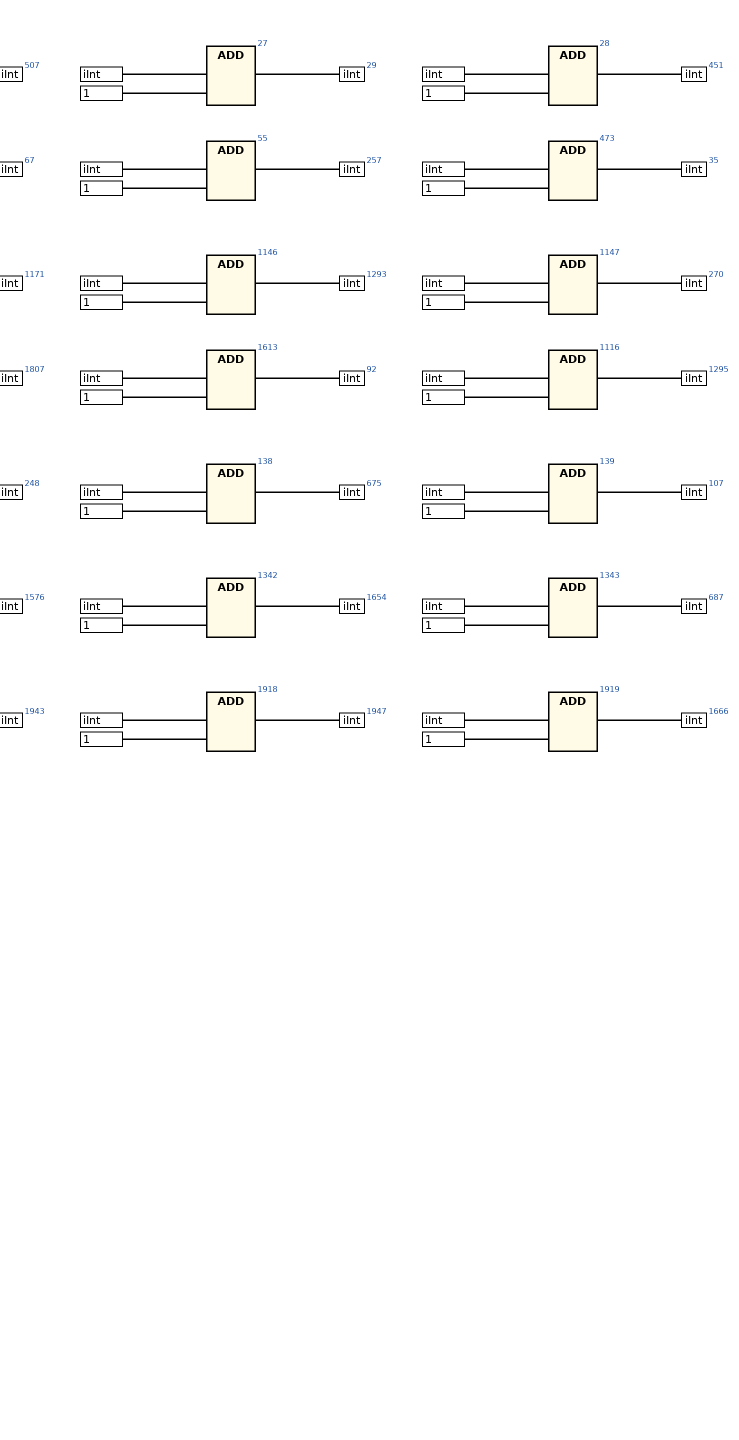
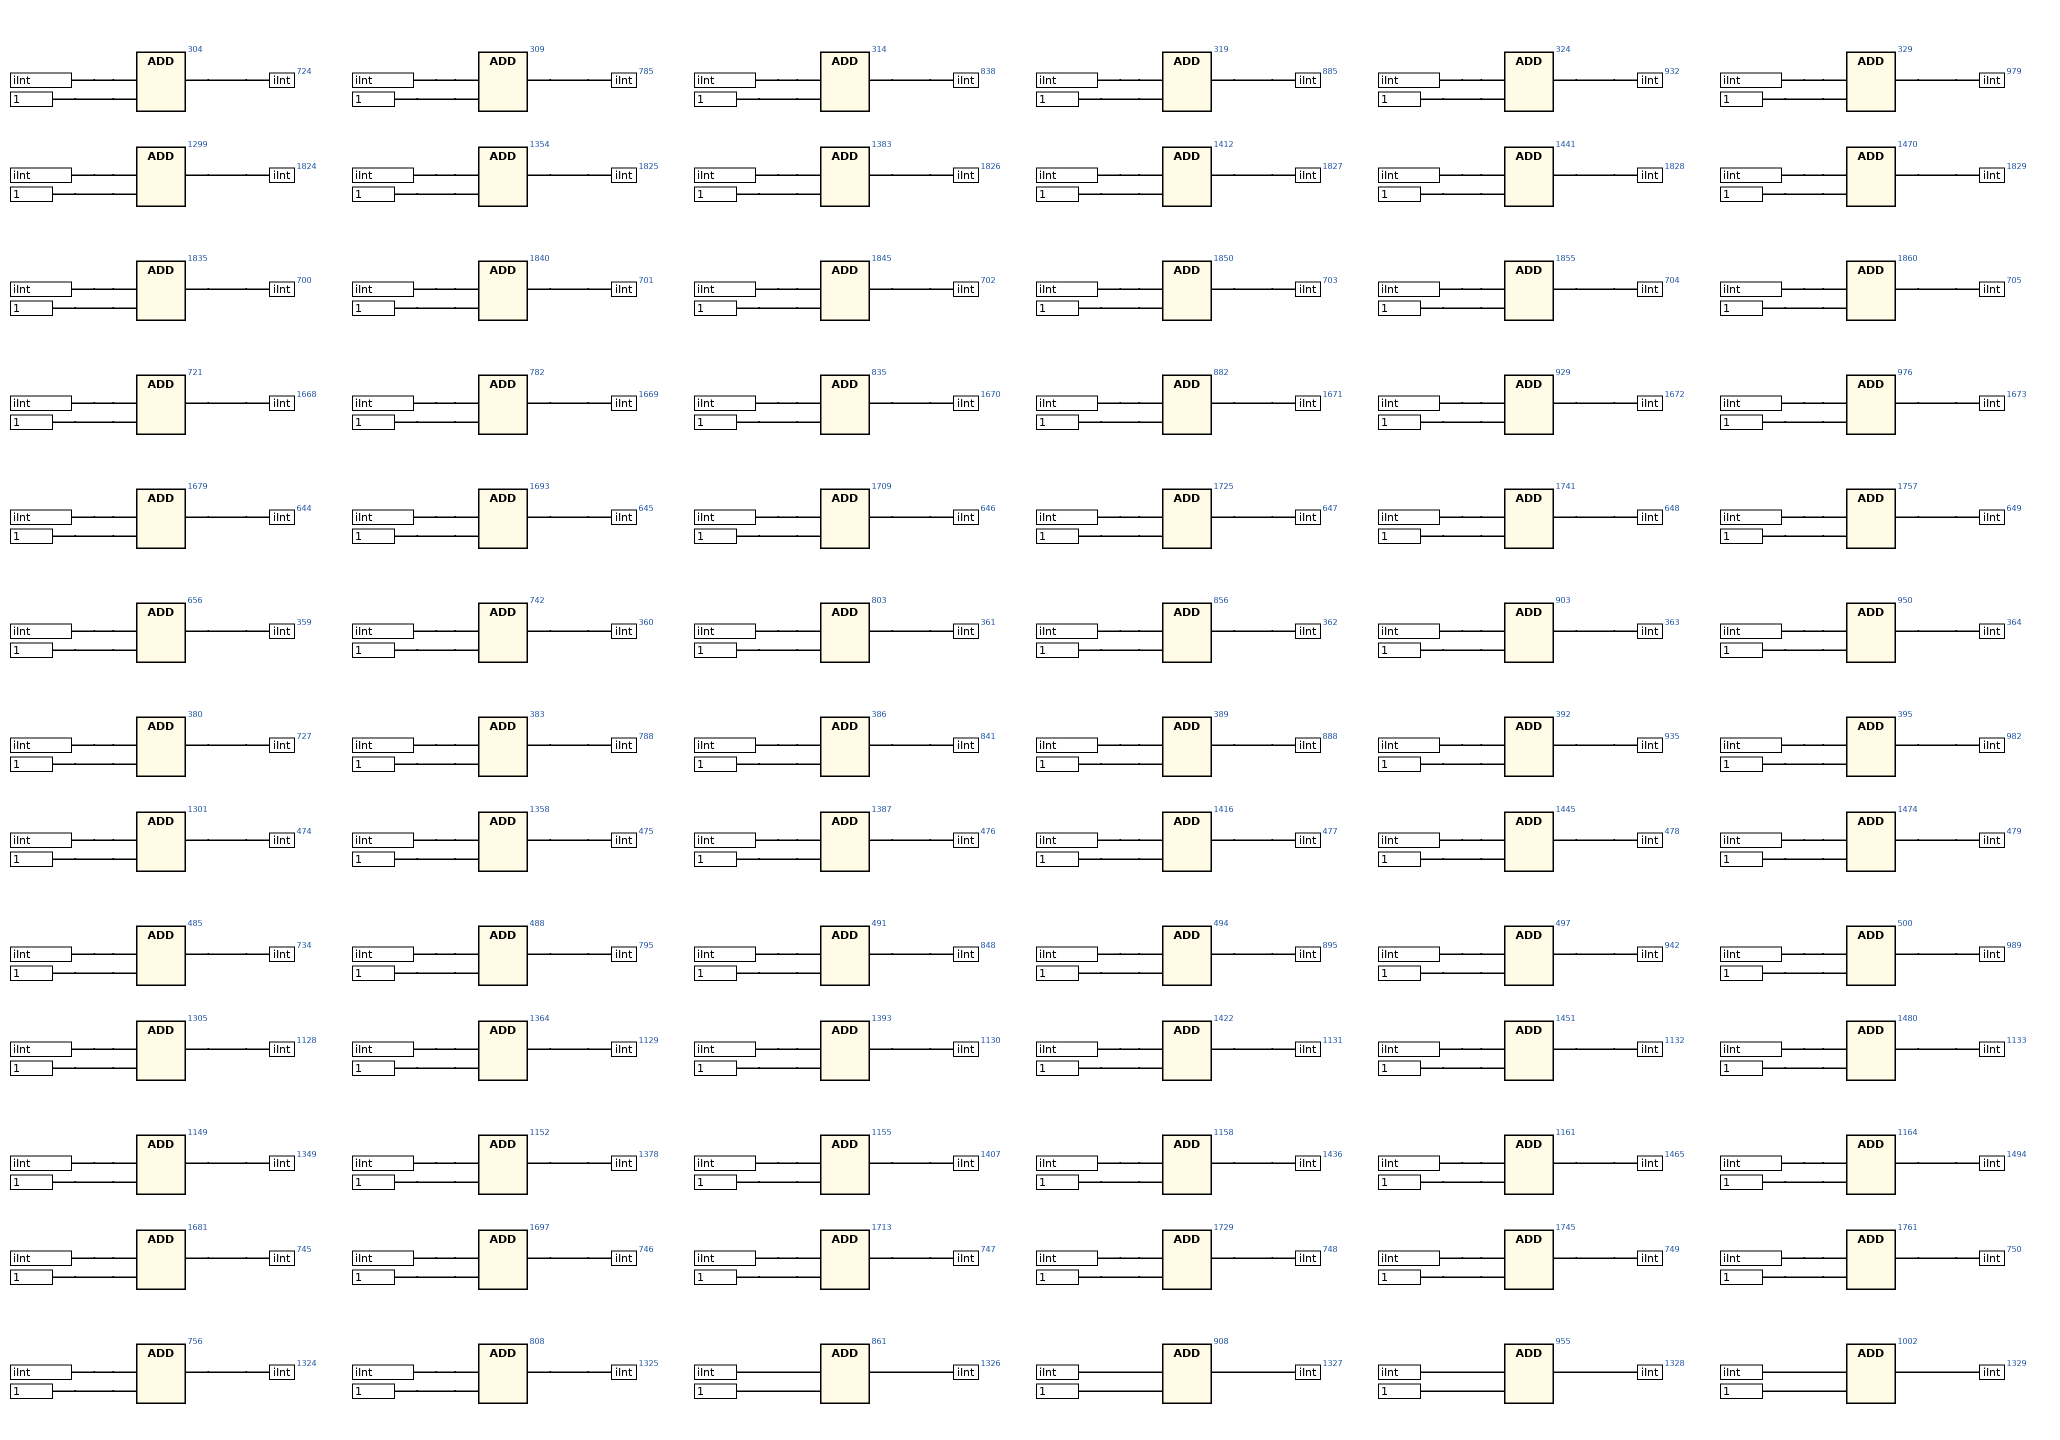
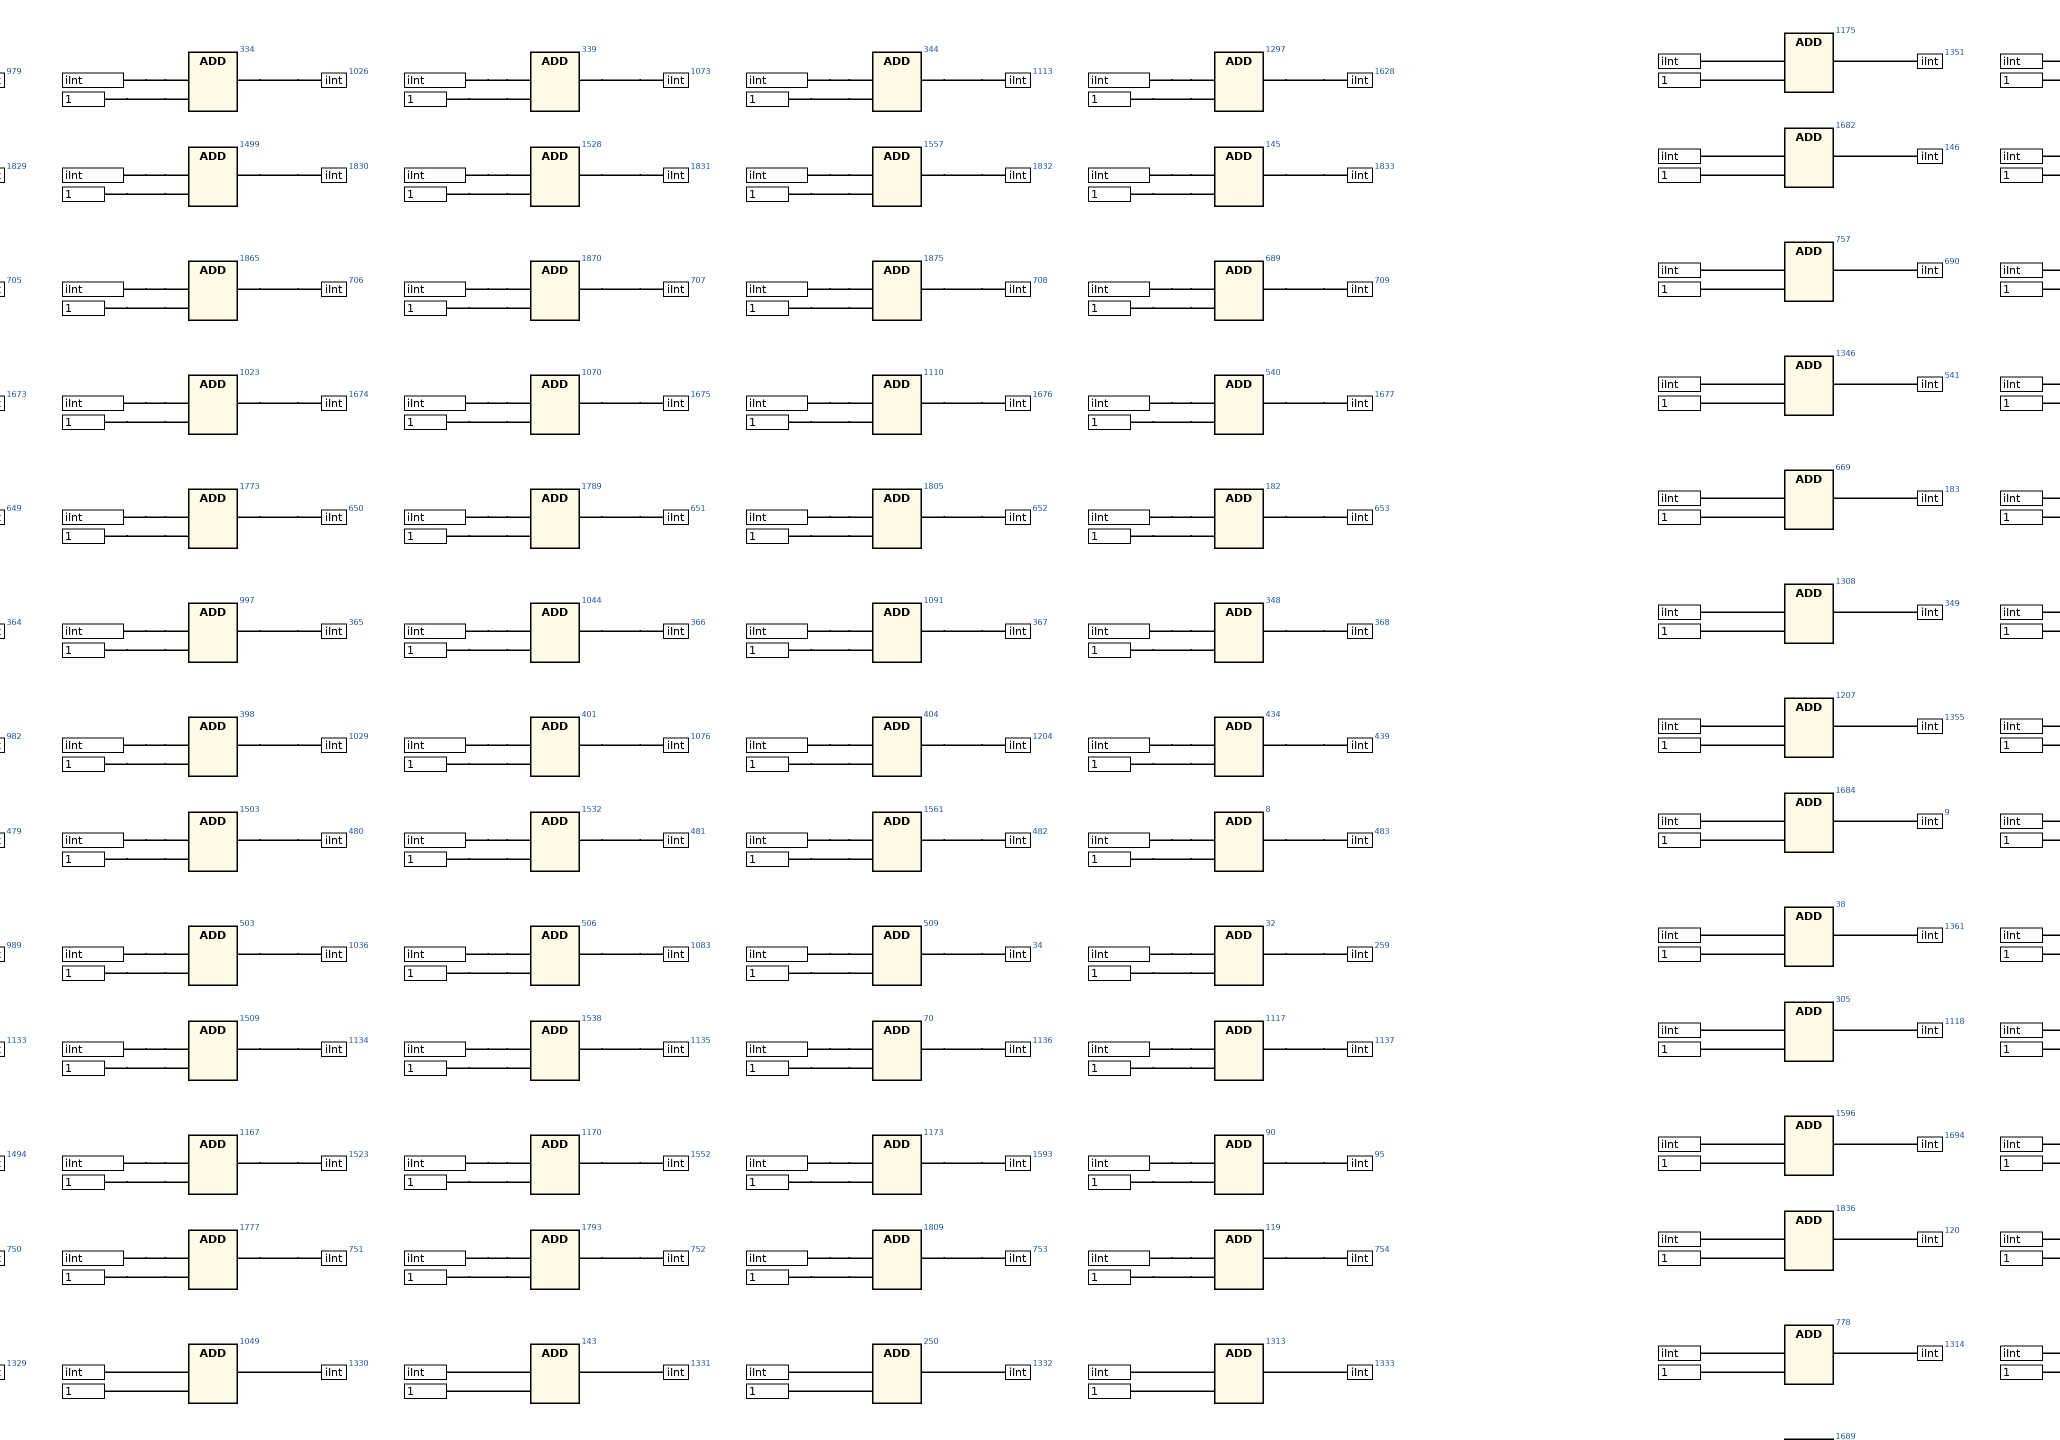
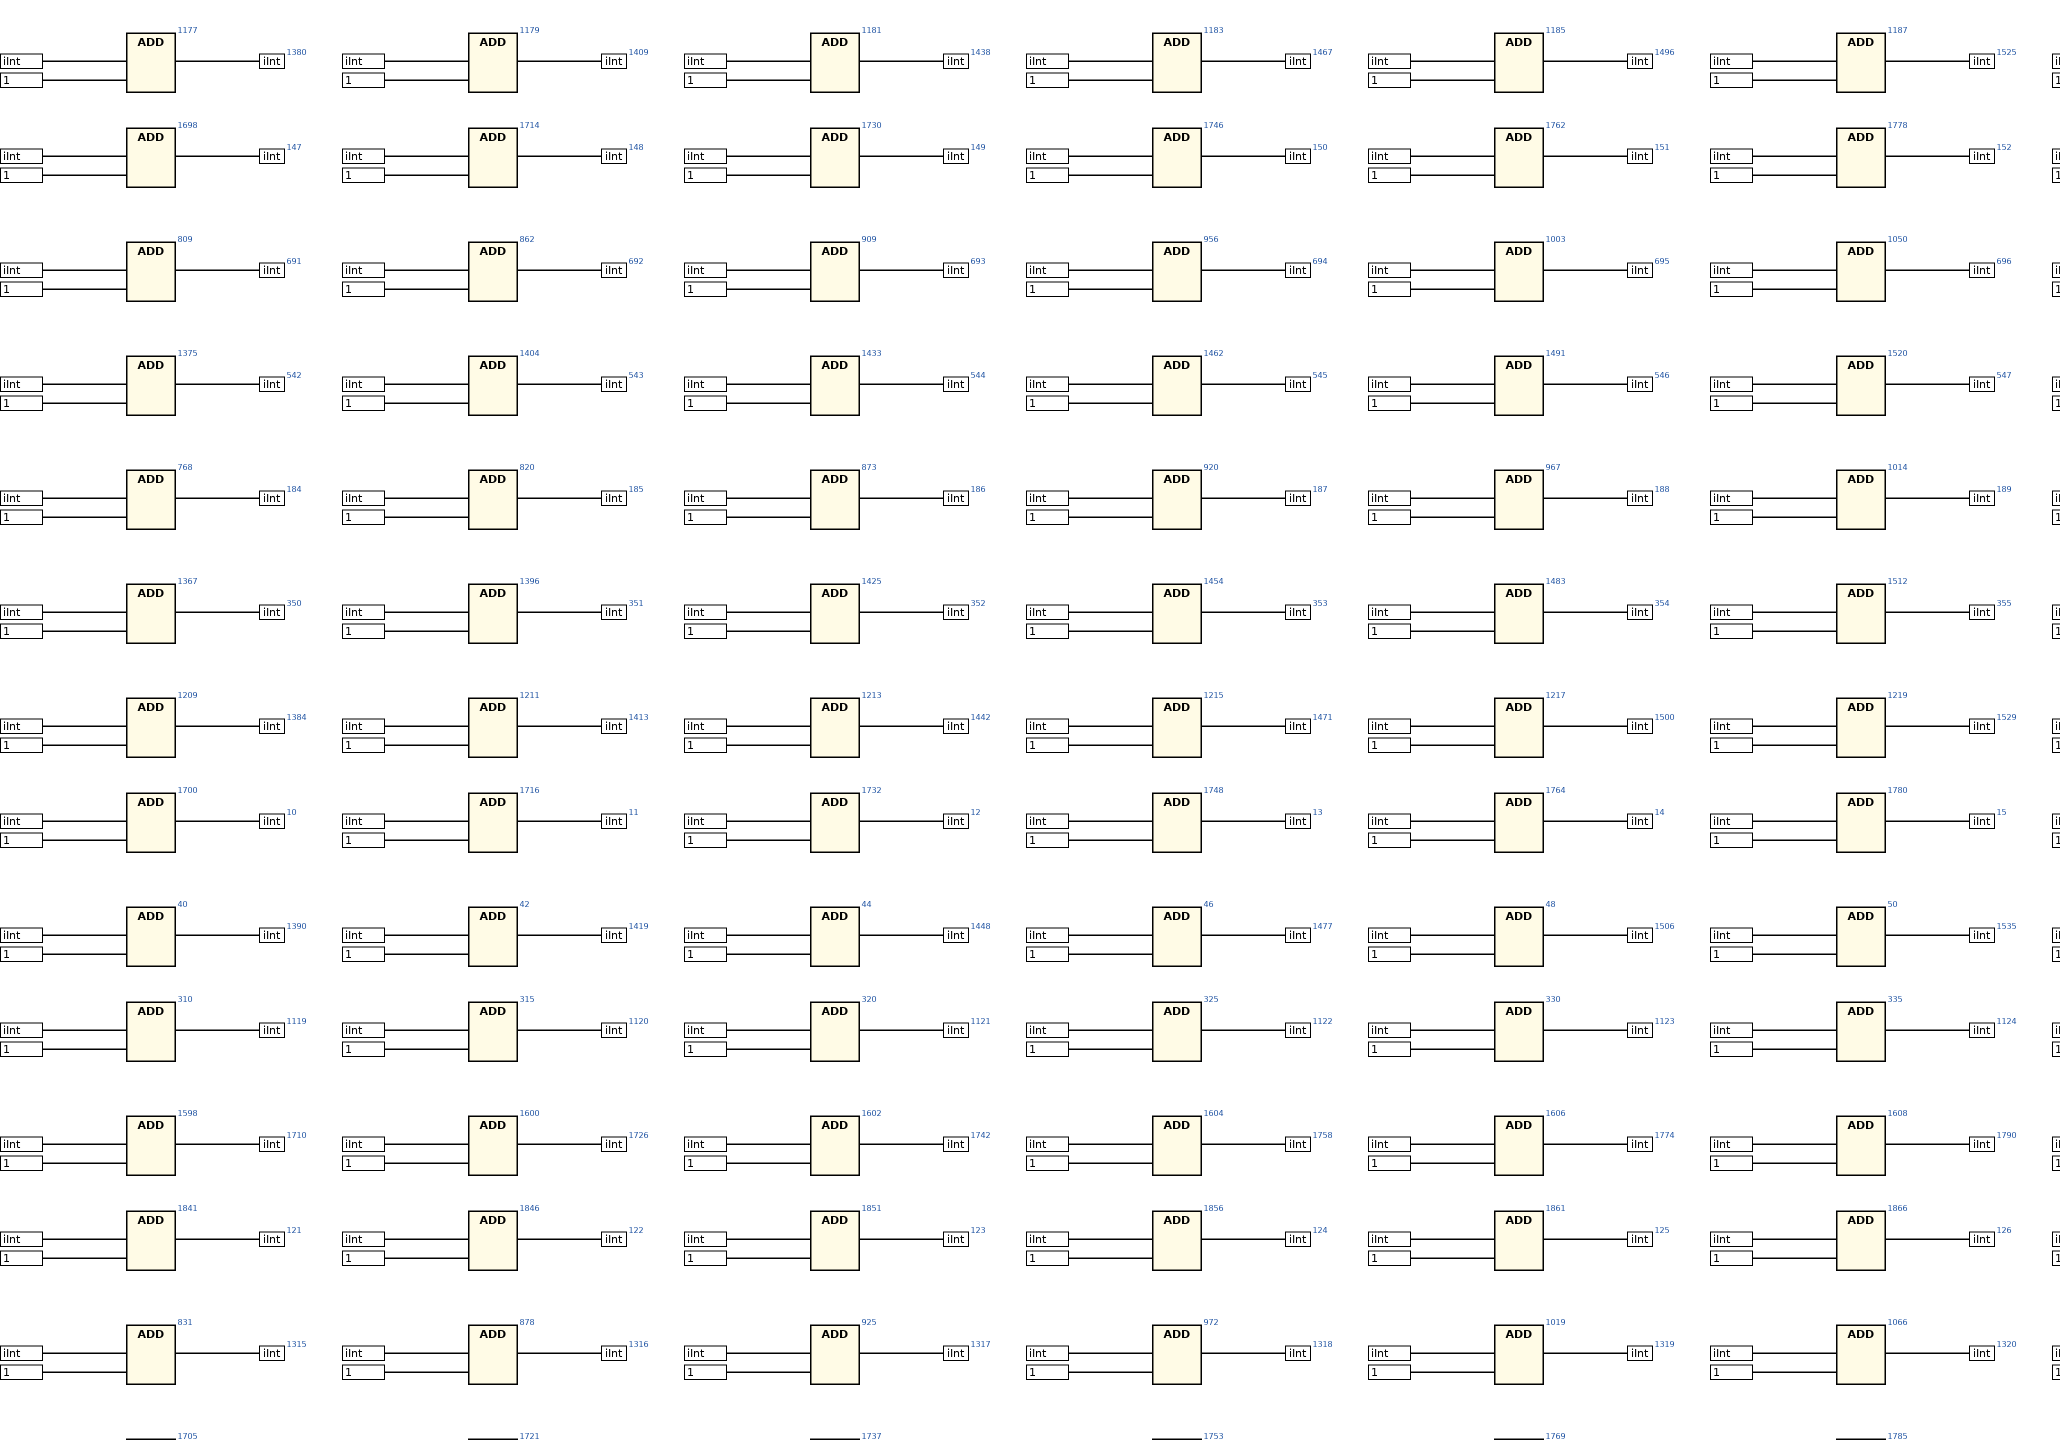
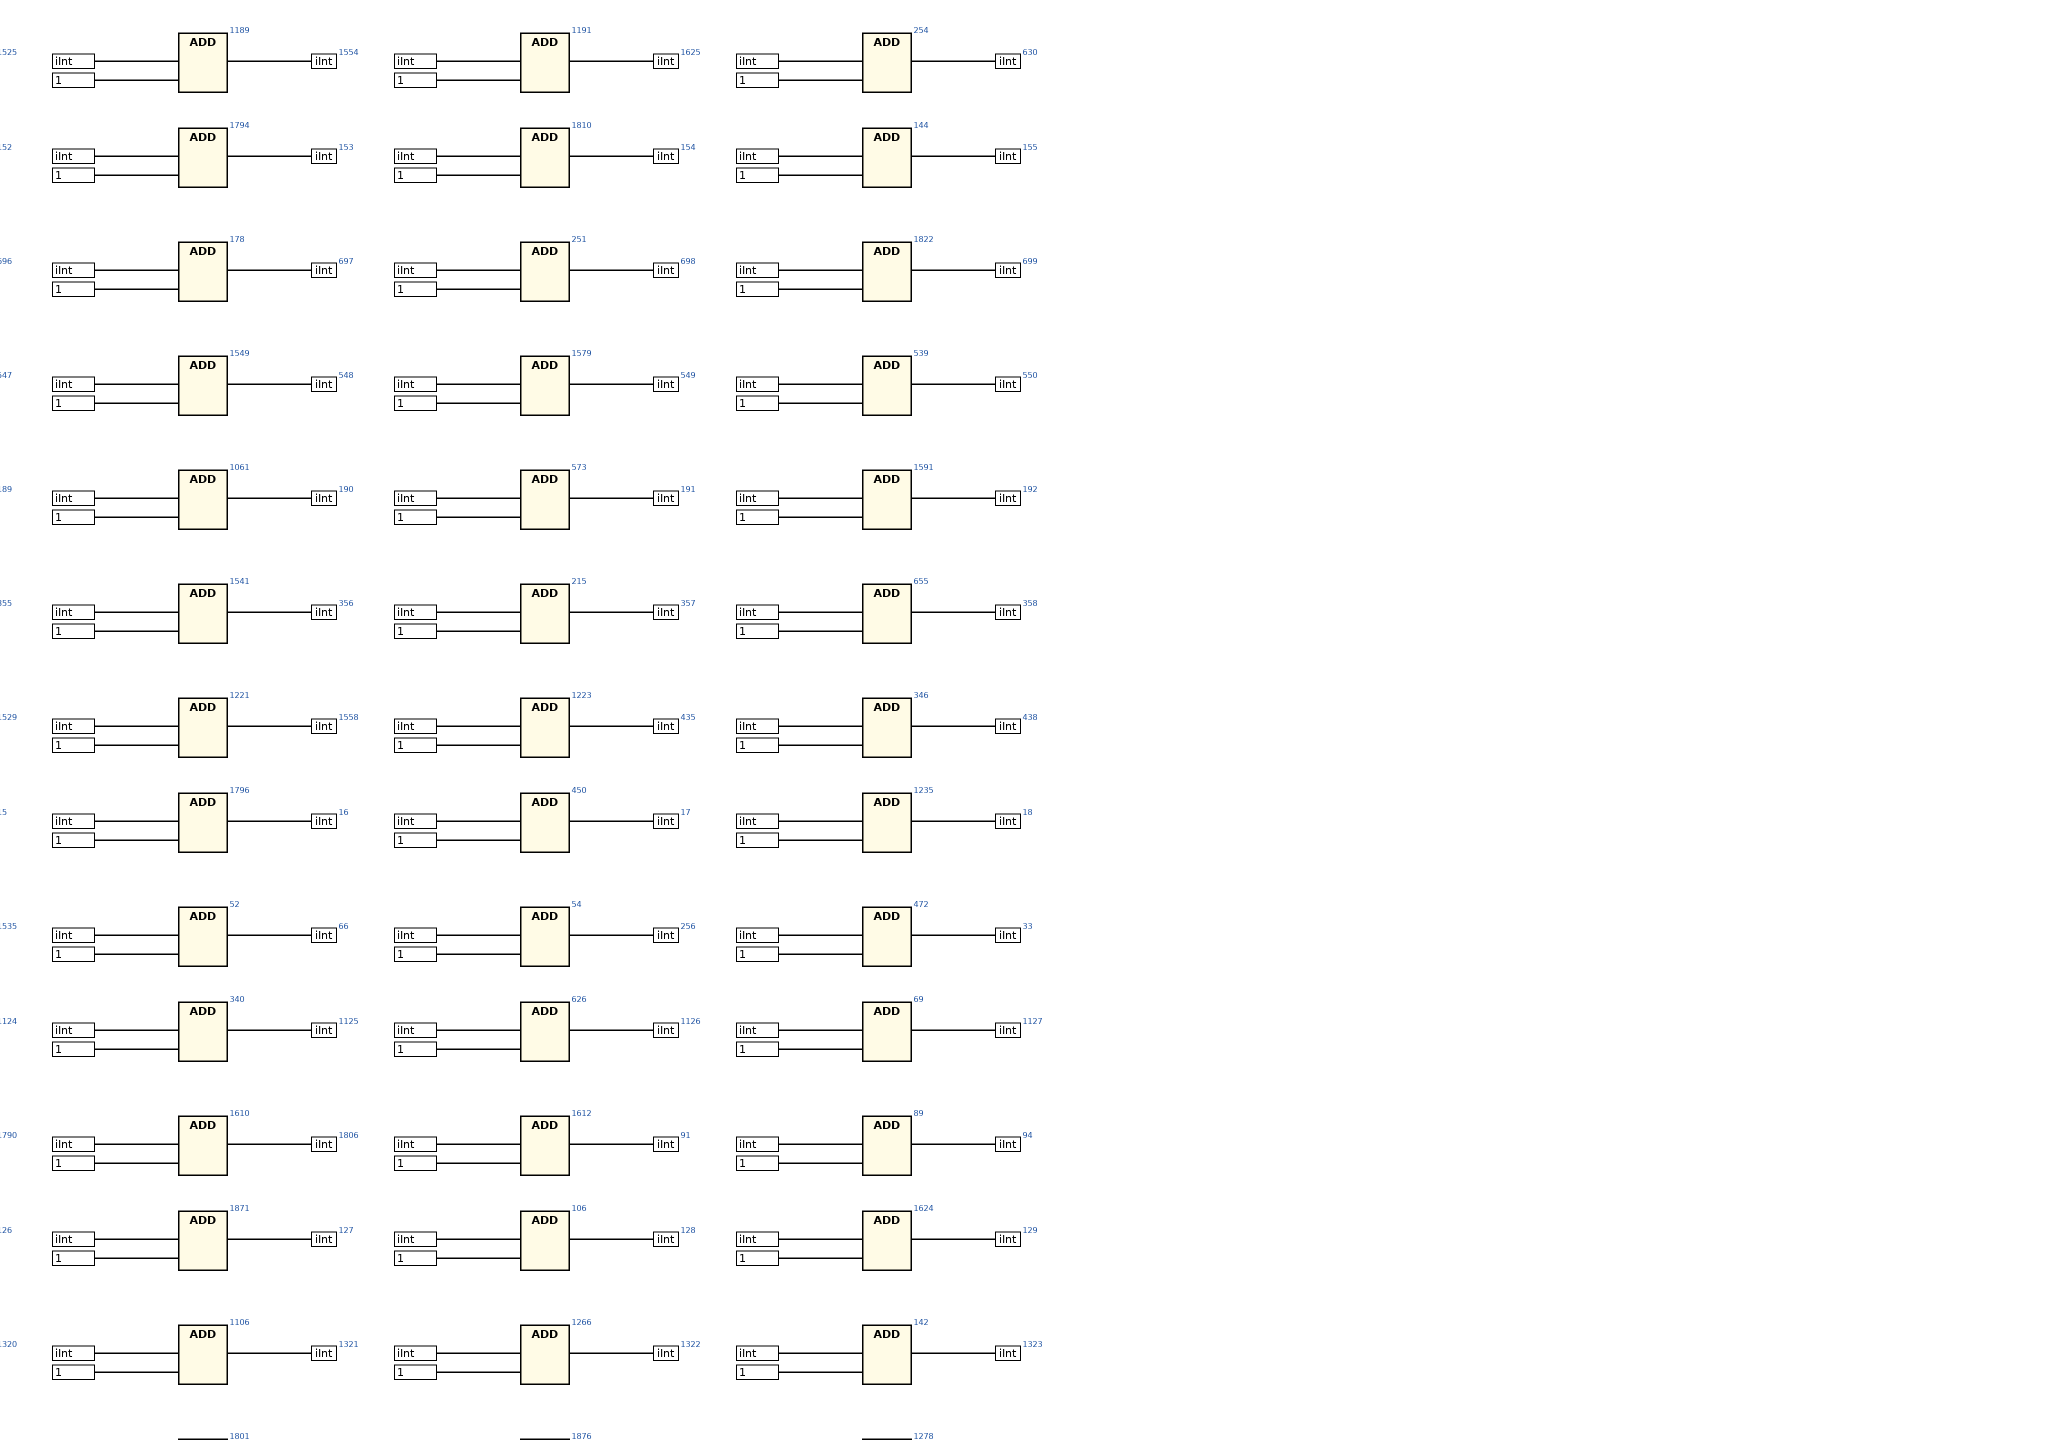
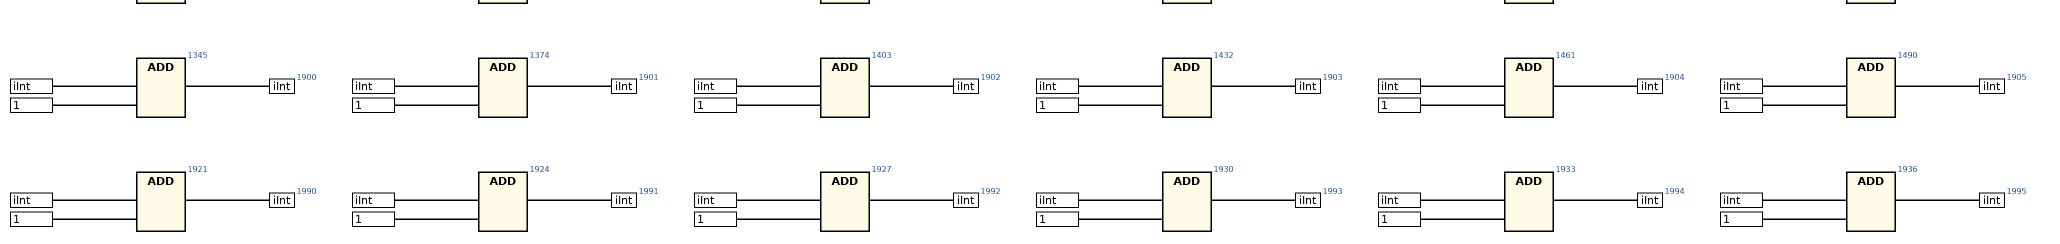
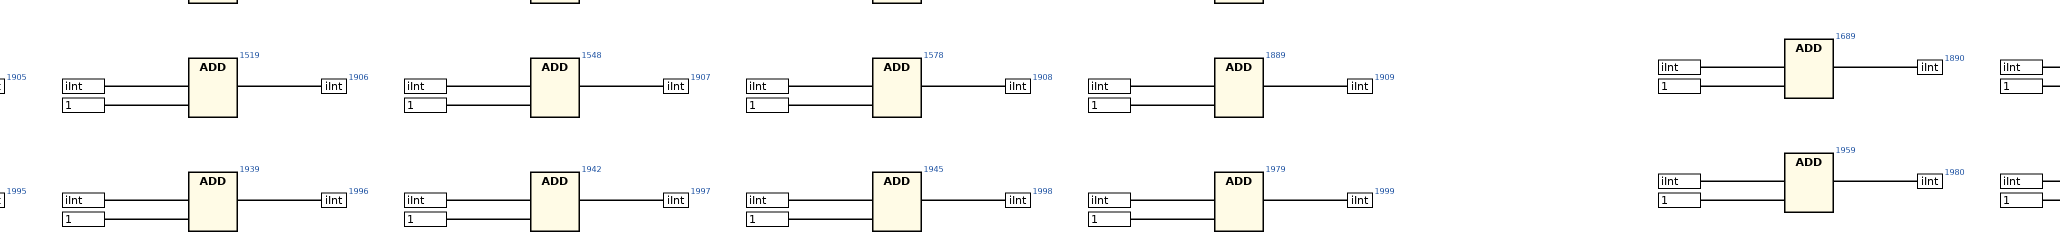
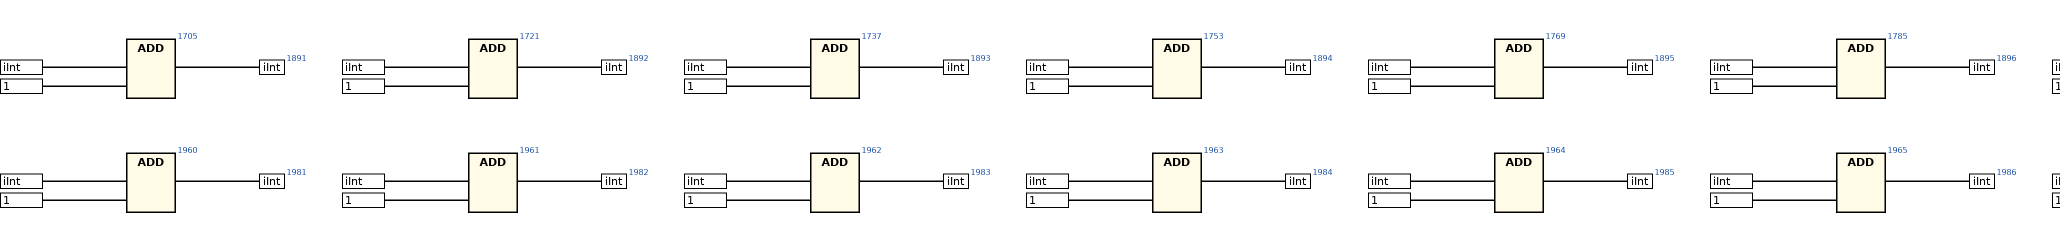
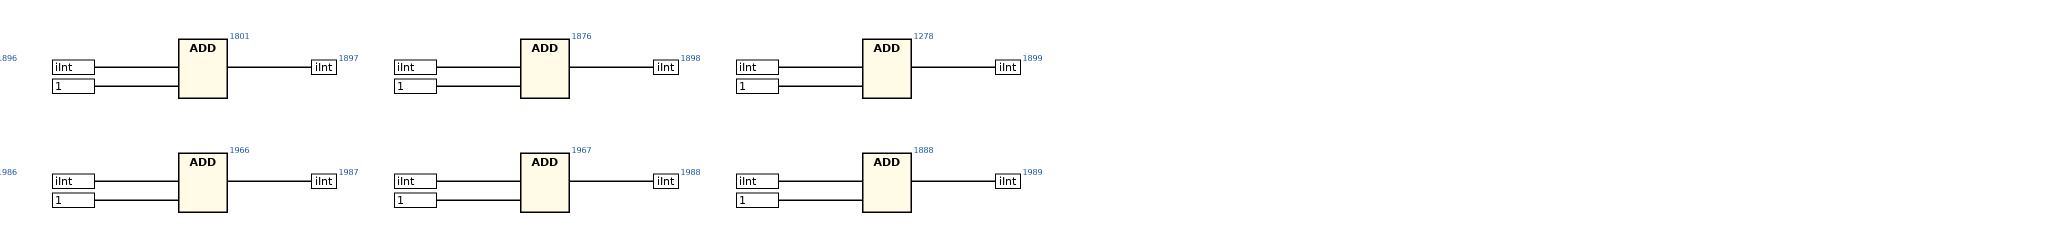
iInt := _w1;
iInt := iInt + 1;
iInt := iInt + 1;
iInt := iInt + 1;
_w2 := iInt + 1;
_w3 := iInt + 1;
iInt := _w4;
iInt := _w5;
iInt := _w6;
iInt := _w7;
iInt := _w8;
iInt := _w9;
iInt := _w10;
iInt := _w11;
iInt := _w12;
iInt := _w13;
_w14 := iInt + 1;
_w15 := iInt + 1;
_w16 := iInt + 1;
_w17 := iInt + 1;
_w18 := iInt + 1;
_w19 := iInt + 1;
_w20 := iInt + 1;
_w21 := iInt + 1;
_w22 := iInt + 1;
iInt := iInt + 1;
_w23 := iInt + 1;
iInt := _w24;
_w25 := iInt + 1;
iInt := _w26;
iInt := _w27;
iInt := _w28;
_w29 := iInt + 1;
iInt := _w23;
_w30 := iInt + 1;
_w31 := iInt + 1;
_w32 := iInt + 1;
_w33 := iInt + 1;
_w34 := iInt + 1;
_w35 := iInt + 1;
_w36 := iInt + 1;
_w37 := iInt + 1;
_w38 := iInt + 1;
_w39 := iInt + 1;
_w40 := iInt + 1;
_w41 := iInt + 1;
_w42 := iInt + 1;
_w43 := iInt + 1;
_w44 := iInt + 1;
_w45 := iInt + 1;
_w46 := iInt + 1;
_w47 := iInt + 1;
iInt := _w48;
iInt := _w49;
iInt := _w50;
iInt := _w51;
iInt := _w52;
iInt := _w53;
iInt := _w54;
iInt := _w55;
iInt := _w56;
iInt := _w29;
iInt := _w44;
iInt := _w45;
_w57 := iInt + 1;
_w58 := iInt + 1;
_w59 := iInt + 1;
_w60 := iInt + 1;
iInt := _w61;
iInt := _w62;
_w63 := iInt + 1;
iInt := _w60;
iInt := _w64;
iInt := _w65;
iInt := _w66;
iInt := _w67;
iInt := _w68;
iInt := _w69;
iInt := _w70;
iInt := _w71;
iInt := _w72;
iInt := _w63;
_w73 := iInt + 1;
iInt := _w74;
_w75 := iInt + 1;
_w76 := iInt + 1;
_w77 := iInt + 1;
iInt := _w78;
iInt := _w79;
_w80 := iInt + 1;
iInt := _w76;
iInt := _w77;
iInt := _w81;
iInt := _w82;
iInt := _w83;
iInt := _w84;
iInt := _w85;
iInt := _w86;
iInt := _w87;
iInt := _w88;
iInt := _w89;
iInt := _w80;
_w90 := iInt + 1;
iInt := _w91;
_w92 := iInt + 1;
iInt := _w93;
iInt := _w94;
iInt := _w95;
iInt := _w96;
iInt := _w97;
iInt := _w98;
iInt := _w99;
iInt := _w100;
iInt := _w101;
iInt := _w92;
_w102 := iInt + 1;
iInt := _w103;
iInt := _w104;
iInt := _w105;
iInt := _w106;
iInt := _w107;
iInt := _w108;
iInt := _w109;
iInt := _w110;
iInt := _w90;
iInt := _w111;
_w112 := iInt + 1;
_w113 := iInt + 1;
_w114 := iInt + 1;
_w115 := iInt + 1;
_w116 := iInt + 1;
_w117 := iInt + 1;
_w118 := iInt + 1;
_w119 := iInt + 1;
_w91 := iInt + 1;
iInt := iInt + 1;
_w120 := iInt + 1;
_w121 := iInt + 1;
_w122 := iInt + 1;
_w123 := iInt + 1;
_w124 := iInt + 1;
iInt := _w125;
iInt := _w126;
iInt := _w127;
iInt := _w128;
iInt := _w129;
iInt := _w130;
iInt := _w131;
iInt := _w132;
iInt := _w133;
iInt := _w123;
_w134 := iInt + 1;
_w135 := iInt + 1;
_w136 := iInt + 1;
_w137 := iInt + 1;
_w138 := iInt + 1;
_w139 := iInt + 1;
_w140 := iInt + 1;
_w141 := iInt + 1;
_w142 := iInt + 1;
iInt := iInt + 1;
_w143 := iInt + 1;
iInt := _w144;
iInt := _w145;
iInt := _w146;
iInt := _w147;
iInt := _w148;
iInt := _w149;
iInt := _w150;
iInt := _w151;
iInt := _w152;
iInt := _w143;
_w153 := iInt + 1;
iInt := _w154;
_w155 := iInt + 1;
iInt := _w156;
_w157 := iInt + 1;
iInt := _w158;
iInt := _w159;
iInt := _w160;
iInt := _w161;
iInt := _w162;
iInt := _w163;
iInt := _w164;
iInt := _w165;
iInt := _w166;
iInt := _w167;
_w168 := iInt + 1;
_w169 := iInt + 1;
_w170 := iInt + 1;
_w171 := iInt + 1;
_w172 := iInt + 1;
_w173 := iInt + 1;
_w174 := iInt + 1;
_w175 := iInt + 1;
_w176 := iInt + 1;
iInt := iInt + 1;
_w177 := iInt + 1;
iInt := _w178;
iInt := _w179;
iInt := _w180;
iInt := _w181;
iInt := _w182;
iInt := _w183;
iInt := _w184;
iInt := _w185;
iInt := _w186;
iInt := _w177;
_w187 := iInt + 1;
iInt := _w188;
_w189 := iInt + 1;
iInt := _w190;
_w191 := iInt + 1;
iInt := _w192;
iInt := _w193;
iInt := _w194;
iInt := _w195;
iInt := _w196;
iInt := _w197;
iInt := _w198;
iInt := _w199;
iInt := _w200;
iInt := _w201;
_w202 := iInt + 1;
_w203 := iInt + 1;
_w204 := iInt + 1;
_w205 := iInt + 1;
_w206 := iInt + 1;
_w207 := iInt + 1;
_w208 := iInt + 1;
_w209 := iInt + 1;
_w210 := iInt + 1;
iInt := iInt + 1;
_w211 := iInt + 1;
iInt := _w210;
iInt := _w212;
iInt := _w213;
iInt := _w214;
iInt := _w215;
_w216 := iInt + 1;
iInt := _w118;
_w217 := iInt + 1;
_w218 := iInt + 1;
_w219 := iInt + 1;
_w220 := iInt + 1;
iInt := _w75;
_w221 := iInt + 1;
_w222 := iInt + 1;
iInt := _w46;
iInt := _w47;
_w223 := iInt + 1;
iInt := _w25;
iInt := _w224;
iInt := _w225;
iInt := _w226;
iInt := _w227;
iInt := _w228;
iInt := _w229;
iInt := _w230;
iInt := _w231;
iInt := _w57;
iInt := _w223;
iInt := _w232;
_w233 := iInt + 1;
_w234 := iInt + 1;
iInt := _w235;
iInt := _w236;
iInt := _w237;
iInt := _w238;
iInt := _w239;
iInt := _w240;
iInt := _w241;
iInt := _w242;
iInt := _w73;
iInt := _w243;
iInt := _w244;
iInt := _w245;
iInt := _w246;
iInt := _w247;
iInt := _w248;
iInt := _w249;
iInt := _w250;
iInt := _w251;
iInt := _w252;
iInt := _w234;
_w253 := iInt + 1;
_w254 := iInt + 1;
_w255 := iInt + 1;
_w256 := iInt + 1;
_w257 := iInt + 1;
_w258 := iInt + 1;
_w259 := iInt + 1;
_w260 := iInt + 1;
_w74 := iInt + 1;
_w261 := iInt + 1;
_w262 := iInt + 1;
_w263 := iInt + 1;
_w264 := iInt + 1;
iInt := iInt + 1;
_w265 := iInt + 1;
_w266 := iInt + 1;
_w267 := iInt + 1;
_w268 := iInt + 1;
iInt := _w253;
_w269 := iInt + 1;
_w270 := iInt + 1;
_w271 := iInt + 1;
_w272 := iInt + 1;
iInt := _w254;
_w273 := iInt + 1;
_w274 := iInt + 1;
_w275 := iInt + 1;
_w276 := iInt + 1;
iInt := _w255;
_w277 := iInt + 1;
_w278 := iInt + 1;
_w279 := iInt + 1;
_w280 := iInt + 1;
iInt := _w256;
_w281 := iInt + 1;
_w282 := iInt + 1;
_w283 := iInt + 1;
_w284 := iInt + 1;
iInt := _w257;
_w285 := iInt + 1;
_w286 := iInt + 1;
_w287 := iInt + 1;
_w288 := iInt + 1;
iInt := _w258;
_w289 := iInt + 1;
_w290 := iInt + 1;
_w291 := iInt + 1;
_w292 := iInt + 1;
iInt := _w259;
_w293 := iInt + 1;
_w294 := iInt + 1;
iInt := _w189;
_w295 := iInt + 1;
_w296 := iInt + 1;
_w297 := iInt + 1;
iInt := _w298;
iInt := _w299;
iInt := _w300;
iInt := _w301;
iInt := _w302;
iInt := _w303;
iInt := _w304;
iInt := _w305;
iInt := _w187;
iInt := _w306;
iInt := _w307;
iInt := _w308;
iInt := _w309;
iInt := _w310;
iInt := _w311;
iInt := _w312;
iInt := _w313;
iInt := _w314;
iInt := _w315;
iInt := _w297;
_w316 := iInt + 1;
_w317 := iInt + 1;
_w318 := iInt + 1;
_w319 := iInt + 1;
_w320 := iInt + 1;
_w321 := iInt + 1;
_w322 := iInt + 1;
_w323 := iInt + 1;
_w188 := iInt + 1;
_w324 := iInt + 1;
_w325 := iInt + 1;
iInt := iInt + 1;
_w326 := iInt + 1;
_w327 := iInt + 1;
iInt := _w316;
_w328 := iInt + 1;
_w329 := iInt + 1;
iInt := _w317;
_w330 := iInt + 1;
_w331 := iInt + 1;
iInt := _w318;
_w332 := iInt + 1;
_w333 := iInt + 1;
iInt := _w319;
_w334 := iInt + 1;
_w335 := iInt + 1;
iInt := _w320;
_w336 := iInt + 1;
_w337 := iInt + 1;
iInt := _w321;
_w338 := iInt + 1;
_w339 := iInt + 1;
iInt := _w322;
_w340 := iInt + 1;
_w341 := iInt + 1;
_w342 := iInt + 1;
_w343 := iInt + 1;
_w344 := iInt + 1;
_w345 := iInt + 1;
_w346 := iInt + 1;
_w347 := iInt + 1;
_w348 := iInt + 1;
_w349 := iInt + 1;
_w350 := iInt + 1;
_w351 := iInt + 1;
_w352 := iInt + 1;
_w353 := iInt + 1;
_w354 := iInt + 1;
_w355 := iInt + 1;
_w356 := iInt + 1;
_w357 := iInt + 1;
_w358 := iInt + 1;
_w359 := iInt + 1;
iInt := _w360;
iInt := _w361;
iInt := _w362;
iInt := _w363;
iInt := _w364;
iInt := _w365;
iInt := _w366;
iInt := _w367;
iInt := _w368;
iInt := _w216;
_w369 := iInt + 1;
_w370 := iInt + 1;
iInt := _w371;
iInt := _w372;
_w373 := iInt + 1;
iInt := _w295;
iInt := _w370;
iInt := _w374;
iInt := _w375;
iInt := _w376;
iInt := _w377;
iInt := _w378;
iInt := _w379;
iInt := _w380;
iInt := _w381;
iInt := _w382;
iInt := _w373;
_w12 := iInt + 1;
iInt := _w22;
_w383 := iInt + 1;
iInt := _w384;
iInt := _w385;
iInt := _w386;
iInt := _w387;
iInt := _w388;
iInt := _w389;
iInt := _w390;
iInt := _w391;
iInt := _w392;
iInt := _w393;
iInt := _w369;
iInt := _w394;
_w395 := iInt + 1;
iInt := _w396;
iInt := _w397;
iInt := _w398;
iInt := _w399;
_w400 := iInt + 1;
iInt := _w383;
_w26 := iInt + 1;
_w28 := iInt + 1;
iInt := _w401;
iInt := _w402;
iInt := _w403;
iInt := _w404;
iInt := _w405;
iInt := _w406;
iInt := _w407;
iInt := _w408;
iInt := _w409;
iInt := _w3;
_w410 := iInt + 1;
_w411 := iInt + 1;
iInt := _w14;
_w412 := iInt + 1;
_w413 := iInt + 1;
iInt := _w15;
_w414 := iInt + 1;
_w415 := iInt + 1;
iInt := _w16;
_w416 := iInt + 1;
_w417 := iInt + 1;
iInt := _w17;
_w418 := iInt + 1;
_w419 := iInt + 1;
iInt := _w18;
_w420 := iInt + 1;
_w421 := iInt + 1;
iInt := _w19;
_w422 := iInt + 1;
_w423 := iInt + 1;
iInt := _w20;
_w424 := iInt + 1;
_w425 := iInt + 1;
iInt := _w21;
_w24 := iInt + 1;
_w27 := iInt + 1;
iInt := _w395;
_w426 := iInt + 1;
_w427 := iInt + 1;
_w428 := iInt + 1;
_w429 := iInt + 1;
_w430 := iInt + 1;
_w431 := iInt + 1;
_w432 := iInt + 1;
_w433 := iInt + 1;
_w434 := iInt + 1;
_w435 := iInt + 1;
_w436 := iInt + 1;
_w437 := iInt + 1;
_w438 := iInt + 1;
_w439 := iInt + 1;
_w440 := iInt + 1;
_w441 := iInt + 1;
_w61 := iInt + 1;
_w62 := iInt + 1;
iInt := _w442;
iInt := _w443;
iInt := _w444;
iInt := _w445;
iInt := _w446;
iInt := _w447;
iInt := _w448;
iInt := _w449;
iInt := _w450;
iInt := _w400;
_w451 := iInt + 1;
_w452 := iInt + 1;
iInt := _w453;
iInt := _w454;
iInt := _w455;
iInt := _w456;
iInt := _w457;
iInt := _w458;
iInt := _w459;
iInt := _w460;
iInt := _w461;
iInt := _w451;
_w462 := iInt + 1;
_w463 := iInt + 1;
_w464 := iInt + 1;
_w465 := iInt + 1;
_w466 := iInt + 1;
_w467 := iInt + 1;
_w468 := iInt + 1;
_w469 := iInt + 1;
_w470 := iInt + 1;
iInt := iInt + 1;
_w471 := iInt + 1;
iInt := _w472;
iInt := _w473;
iInt := _w474;
iInt := _w475;
iInt := _w476;
iInt := _w477;
iInt := _w478;
iInt := _w479;
iInt := _w480;
iInt := _w471;
_w166 := iInt + 1;
iInt := _w176;
_w481 := iInt + 1;
iInt := _w482;
iInt := _w483;
iInt := _w484;
iInt := _w485;
iInt := _w486;
iInt := _w487;
iInt := _w488;
iInt := _w489;
iInt := _w490;
iInt := _w481;
_w491 := iInt + 1;
_w492 := iInt + 1;
_w493 := iInt + 1;
_w494 := iInt + 1;
_w495 := iInt + 1;
_w496 := iInt + 1;
_w497 := iInt + 1;
_w498 := iInt + 1;
_w1 := iInt + 1;
iInt := iInt + 1;
_w499 := iInt + 1;
iInt := _w500;
iInt := _w501;
iInt := _w502;
iInt := _w503;
iInt := _w504;
iInt := _w505;
iInt := _w506;
iInt := _w507;
iInt := _w508;
iInt := _w499;
_w509 := iInt + 1;
_w360 := iInt + 1;
_w442 := iInt + 1;
_w482 := iInt + 1;
_w500 := iInt + 1;
_w201 := iInt + 1;
_w510 := iInt + 1;
_w511 := iInt + 1;
iInt := _w512;
iInt := _w513;
iInt := _w514;
iInt := _w515;
iInt := _w516;
iInt := _w517;
iInt := _w518;
iInt := _w519;
iInt := _w155;
iInt := _w220;
_w520 := iInt + 1;
_w521 := iInt + 1;
iInt := _w260;
_w522 := iInt + 1;
iInt := _w221;
iInt := _w222;
_w523 := iInt + 1;
iInt := _w323;
_w524 := iInt + 1;
iInt := _w296;
_w525 := iInt + 1;
_w526 := iInt + 1;
_w527 := iInt + 1;
_w528 := iInt + 1;
_w48 := iInt + 1;
_w64 := iInt + 1;
_w243 := iInt + 1;
_w244 := iInt + 1;
iInt := _w529;
iInt := _w530;
iInt := _w531;
iInt := _w532;
iInt := _w533;
iInt := _w534;
iInt := _w535;
iInt := _w536;
iInt := _w537;
iInt := _w157;
_w178 := iInt + 1;
_w306 := iInt + 1;
_w307 := iInt + 1;
_w192 := iInt + 1;
_w538 := iInt + 1;
_w512 := iInt + 1;
iInt := _w539;
iInt := _w540;
iInt := _w541;
iInt := _w542;
_w361 := iInt + 1;
iInt := _w543;
iInt := _w544;
iInt := _w545;
_w443 := iInt + 1;
_w158 := iInt + 1;
_w483 := iInt + 1;
iInt := _w491;
_w501 := iInt + 1;
_w546 := iInt + 1;
_w547 := iInt + 1;
iInt := _w119;
_w548 := iInt + 1;
iInt := _w549;
iInt := _w550;
iInt := _w551;
iInt := _w552;
iInt := _w553;
iInt := _w554;
iInt := _w555;
iInt := _w120;
iInt := _w217;
iInt := _w548;
iInt := _w556;
_w557 := iInt + 1;
_w558 := iInt + 1;
iInt := _w559;
iInt := _w560;
iInt := _w561;
iInt := _w562;
iInt := _w563;
iInt := _w564;
iInt := _w565;
iInt := _w153;
iInt := _w219;
iInt := _w566;
iInt := _w567;
iInt := _w568;
iInt := _w569;
iInt := _w570;
iInt := _w571;
iInt := _w572;
iInt := _w573;
iInt := _w574;
iInt := _w575;
iInt := _w558;
_w576 := iInt + 1;
_w577 := iInt + 1;
_w578 := iInt + 1;
_w579 := iInt + 1;
_w580 := iInt + 1;
_w581 := iInt + 1;
_w582 := iInt + 1;
_w583 := iInt + 1;
_w584 := iInt + 1;
_w154 := iInt + 1;
_w585 := iInt + 1;
_w586 := iInt + 1;
iInt := _w233;
iInt := _w261;
iInt := _w262;
_w587 := iInt + 1;
iInt := _w324;
iInt := _w325;
_w588 := iInt + 1;
iInt := _w342;
iInt := _w343;
_w589 := iInt + 1;
_w590 := iInt + 1;
iInt := _w410;
iInt := _w411;
_w49 := iInt + 1;
iInt := _w426;
iInt := _w427;
_w65 := iInt + 1;
_w245 := iInt + 1;
iInt := _w168;
_w179 := iInt + 1;
_w308 := iInt + 1;
_w193 := iInt + 1;
_w591 := iInt + 1;
iInt := _w592;
iInt := _w593;
iInt := _w594;
iInt := _w595;
iInt := _w596;
iInt := _w597;
iInt := _w598;
iInt := _w599;
iInt := _w600;
iInt := _w102;
_w549 := iInt + 1;
_w601 := iInt + 1;
_w559 := iInt + 1;
_w513 := iInt + 1;
iInt := _w602;
iInt := _w603;
iInt := _w604;
iInt := _w605;
_w362 := iInt + 1;
iInt := _w606;
iInt := _w607;
iInt := _w608;
_w444 := iInt + 1;
_w159 := iInt + 1;
_w484 := iInt + 1;
iInt := _w492;
_w502 := iInt + 1;
_w609 := iInt + 1;
iInt := iInt + 1;
iInt := iInt + 1;
_w610 := iInt + 1;
_w611 := iInt + 1;
_w612 := iInt + 1;
iInt := _w576;
_w613 := iInt + 1;
_w614 := iInt + 1;
iInt := _w264;
iInt := _w265;
iInt := _w266;
_w615 := iInt + 1;
iInt := _w326;
iInt := _w327;
_w616 := iInt + 1;
iInt := _w344;
iInt := _w345;
_w617 := iInt + 1;
_w618 := iInt + 1;
iInt := _w412;
iInt := _w413;
_w50 := iInt + 1;
iInt := _w428;
iInt := _w429;
_w66 := iInt + 1;
_w246 := iInt + 1;
iInt := _w169;
_w180 := iInt + 1;
_w309 := iInt + 1;
_w194 := iInt + 1;
_w619 := iInt + 1;
iInt := _w112;
_w550 := iInt + 1;
_w620 := iInt + 1;
_w560 := iInt + 1;
_w514 := iInt + 1;
iInt := _w621;
iInt := _w622;
iInt := _w623;
iInt := _w624;
_w363 := iInt + 1;
iInt := _w625;
iInt := _w626;
iInt := _w627;
_w445 := iInt + 1;
_w160 := iInt + 1;
_w485 := iInt + 1;
iInt := _w493;
_w503 := iInt + 1;
_w628 := iInt + 1;
_w629 := iInt + 1;
iInt := _w2;
iInt := _w511;
iInt := _w547;
iInt := _w610;
iInt := _w629;
_w630 := iInt + 1;
_w631 := iInt + 1;
iInt := _w577;
_w632 := iInt + 1;
_w633 := iInt + 1;
iInt := _w268;
iInt := _w269;
iInt := _w270;
_w634 := iInt + 1;
iInt := _w328;
iInt := _w329;
_w635 := iInt + 1;
iInt := _w346;
iInt := _w347;
_w636 := iInt + 1;
_w637 := iInt + 1;
iInt := _w414;
iInt := _w415;
_w51 := iInt + 1;
iInt := _w430;
iInt := _w431;
_w67 := iInt + 1;
_w247 := iInt + 1;
iInt := _w170;
_w181 := iInt + 1;
_w310 := iInt + 1;
_w195 := iInt + 1;
_w638 := iInt + 1;
iInt := _w113;
_w551 := iInt + 1;
_w639 := iInt + 1;
_w561 := iInt + 1;
_w515 := iInt + 1;
iInt := _w640;
iInt := _w641;
iInt := _w642;
iInt := _w643;
_w364 := iInt + 1;
iInt := _w644;
iInt := _w645;
iInt := _w646;
_w446 := iInt + 1;
_w161 := iInt + 1;
_w486 := iInt + 1;
iInt := _w494;
_w504 := iInt + 1;
_w647 := iInt + 1;
_w648 := iInt + 1;
_w649 := iInt + 1;
iInt := _w578;
_w650 := iInt + 1;
_w651 := iInt + 1;
iInt := _w272;
iInt := _w273;
iInt := _w274;
_w652 := iInt + 1;
iInt := _w330;
iInt := _w331;
_w653 := iInt + 1;
iInt := _w348;
iInt := _w349;
_w654 := iInt + 1;
_w655 := iInt + 1;
iInt := _w416;
iInt := _w417;
_w52 := iInt + 1;
iInt := _w432;
iInt := _w433;
_w68 := iInt + 1;
_w248 := iInt + 1;
iInt := _w171;
_w182 := iInt + 1;
_w311 := iInt + 1;
_w196 := iInt + 1;
_w656 := iInt + 1;
iInt := _w114;
_w552 := iInt + 1;
_w657 := iInt + 1;
_w562 := iInt + 1;
_w516 := iInt + 1;
iInt := _w658;
iInt := _w659;
iInt := _w660;
iInt := _w661;
_w365 := iInt + 1;
iInt := _w662;
iInt := _w663;
iInt := _w664;
_w447 := iInt + 1;
_w162 := iInt + 1;
_w487 := iInt + 1;
iInt := _w495;
_w505 := iInt + 1;
_w665 := iInt + 1;
_w666 := iInt + 1;
_w667 := iInt + 1;
iInt := _w579;
_w668 := iInt + 1;
_w669 := iInt + 1;
iInt := _w276;
iInt := _w277;
iInt := _w278;
_w670 := iInt + 1;
iInt := _w332;
iInt := _w333;
_w671 := iInt + 1;
iInt := _w350;
iInt := _w351;
_w672 := iInt + 1;
_w673 := iInt + 1;
iInt := _w418;
iInt := _w419;
_w53 := iInt + 1;
iInt := _w434;
iInt := _w435;
_w69 := iInt + 1;
_w249 := iInt + 1;
iInt := _w172;
_w183 := iInt + 1;
_w312 := iInt + 1;
_w197 := iInt + 1;
_w674 := iInt + 1;
iInt := _w115;
_w553 := iInt + 1;
_w675 := iInt + 1;
_w563 := iInt + 1;
_w517 := iInt + 1;
iInt := _w676;
iInt := _w677;
iInt := _w678;
iInt := _w679;
_w366 := iInt + 1;
iInt := _w680;
iInt := _w681;
iInt := _w682;
_w448 := iInt + 1;
_w163 := iInt + 1;
_w488 := iInt + 1;
iInt := _w496;
_w506 := iInt + 1;
_w683 := iInt + 1;
_w684 := iInt + 1;
_w685 := iInt + 1;
iInt := _w580;
_w686 := iInt + 1;
_w687 := iInt + 1;
iInt := _w280;
iInt := _w281;
iInt := _w282;
_w688 := iInt + 1;
iInt := _w334;
iInt := _w335;
_w689 := iInt + 1;
iInt := _w352;
iInt := _w353;
_w690 := iInt + 1;
_w691 := iInt + 1;
iInt := _w420;
iInt := _w421;
_w54 := iInt + 1;
iInt := _w436;
iInt := _w437;
_w70 := iInt + 1;
_w250 := iInt + 1;
iInt := _w173;
_w184 := iInt + 1;
_w313 := iInt + 1;
_w198 := iInt + 1;
_w692 := iInt + 1;
iInt := _w116;
_w554 := iInt + 1;
_w693 := iInt + 1;
_w564 := iInt + 1;
_w518 := iInt + 1;
iInt := _w694;
iInt := _w695;
iInt := _w696;
iInt := _w697;
_w367 := iInt + 1;
iInt := _w698;
iInt := _w699;
iInt := _w700;
_w449 := iInt + 1;
_w164 := iInt + 1;
_w489 := iInt + 1;
iInt := _w497;
_w507 := iInt + 1;
_w701 := iInt + 1;
_w702 := iInt + 1;
_w703 := iInt + 1;
iInt := _w581;
_w704 := iInt + 1;
_w705 := iInt + 1;
iInt := _w284;
iInt := _w285;
iInt := _w286;
_w706 := iInt + 1;
iInt := _w336;
iInt := _w337;
_w707 := iInt + 1;
iInt := _w354;
iInt := _w355;
_w708 := iInt + 1;
_w709 := iInt + 1;
iInt := _w422;
iInt := _w423;
_w55 := iInt + 1;
iInt := _w438;
iInt := _w439;
_w71 := iInt + 1;
_w251 := iInt + 1;
iInt := _w174;
_w185 := iInt + 1;
_w314 := iInt + 1;
_w199 := iInt + 1;
_w710 := iInt + 1;
iInt := _w117;
_w555 := iInt + 1;
_w711 := iInt + 1;
_w565 := iInt + 1;
_w519 := iInt + 1;
iInt := _w712;
iInt := _w713;
iInt := _w714;
iInt := _w715;
_w368 := iInt + 1;
iInt := _w716;
iInt := _w717;
iInt := _w718;
_w450 := iInt + 1;
_w165 := iInt + 1;
_w490 := iInt + 1;
iInt := _w498;
_w508 := iInt + 1;
_w719 := iInt + 1;
_w720 := iInt + 1;
_w721 := iInt + 1;
iInt := _w582;
_w722 := iInt + 1;
_w723 := iInt + 1;
iInt := _w288;
iInt := _w289;
iInt := _w290;
_w724 := iInt + 1;
iInt := _w338;
iInt := _w339;
_w725 := iInt + 1;
iInt := _w356;
iInt := _w357;
_w726 := iInt + 1;
_w727 := iInt + 1;
iInt := _w424;
iInt := _w425;
_w56 := iInt + 1;
iInt := _w440;
iInt := _w441;
_w72 := iInt + 1;
_w252 := iInt + 1;
iInt := _w175;
_w186 := iInt + 1;
_w315 := iInt + 1;
_w200 := iInt + 1;
_w728 := iInt + 1;
iInt := _w509;
iInt := _w538;
iInt := _w591;
iInt := _w619;
iInt := _w638;
iInt := _w656;
iInt := _w674;
iInt := _w692;
iInt := _w710;
iInt := _w728;
_w213 := iInt + 1;
_w215 := iInt + 1;
_w729 := iInt + 1;
_w730 := iInt + 1;
iInt := _w583;
_w731 := iInt + 1;
_w732 := iInt + 1;
iInt := _w292;
iInt := _w293;
iInt := _w294;
_w733 := iInt + 1;
iInt := _w521;
_w734 := iInt + 1;
_w735 := iInt + 1;
iInt := _w263;
iInt := _w267;
iInt := _w271;
iInt := _w275;
iInt := _w279;
iInt := _w283;
iInt := _w287;
iInt := _w291;
iInt := _w520;
iInt := _w58;
iInt := _w736;
iInt := _w737;
iInt := _w738;
iInt := _w739;
iInt := _w740;
iInt := _w741;
iInt := _w742;
iInt := _w743;
iInt := _w59;
iInt := _w735;
_w744 := iInt + 1;
_w745 := iInt + 1;
_w746 := iInt + 1;
_w747 := iInt + 1;
_w748 := iInt + 1;
_w749 := iInt + 1;
_w750 := iInt + 1;
_w751 := iInt + 1;
_w232 := iInt + 1;
_w752 := iInt + 1;
_w753 := iInt + 1;
iInt := iInt + 1;
_w754 := iInt + 1;
_w755 := iInt + 1;
iInt := _w744;
_w756 := iInt + 1;
_w757 := iInt + 1;
iInt := _w745;
_w758 := iInt + 1;
_w759 := iInt + 1;
iInt := _w746;
_w760 := iInt + 1;
_w761 := iInt + 1;
iInt := _w747;
_w762 := iInt + 1;
_w763 := iInt + 1;
iInt := _w748;
_w764 := iInt + 1;
_w765 := iInt + 1;
iInt := _w749;
_w766 := iInt + 1;
_w767 := iInt + 1;
iInt := _w750;
_w768 := iInt + 1;
_w769 := iInt + 1;
iInt := _w522;
_w770 := iInt + 1;
_w771 := iInt + 1;
_w772 := iInt + 1;
_w773 := iInt + 1;
_w774 := iInt + 1;
_w775 := iInt + 1;
_w776 := iInt + 1;
_w777 := iInt + 1;
_w778 := iInt + 1;
_w779 := iInt + 1;
_w780 := iInt + 1;
_w781 := iInt + 1;
_w782 := iInt + 1;
_w783 := iInt + 1;
_w784 := iInt + 1;
_w785 := iInt + 1;
_w786 := iInt + 1;
_w787 := iInt + 1;
iInt := _w523;
iInt := _w587;
iInt := _w615;
iInt := _w634;
iInt := _w652;
iInt := _w670;
iInt := _w688;
iInt := _w706;
iInt := _w724;
iInt := _w733;
iInt := _w340;
iInt := _w341;
_w788 := iInt + 1;
iInt := _w524;
_w789 := iInt + 1;
_w790 := iInt + 1;
_w791 := iInt + 1;
_w792 := iInt + 1;
_w793 := iInt + 1;
_w794 := iInt + 1;
_w795 := iInt + 1;
_w796 := iInt + 1;
_w797 := iInt + 1;
_w798 := iInt + 1;
_w799 := iInt + 1;
_w800 := iInt + 1;
_w801 := iInt + 1;
_w802 := iInt + 1;
_w803 := iInt + 1;
_w804 := iInt + 1;
_w371 := iInt + 1;
_w372 := iInt + 1;
iInt := _w525;
iInt := _w588;
iInt := _w616;
iInt := _w635;
iInt := _w653;
iInt := _w671;
iInt := _w689;
iInt := _w707;
iInt := _w725;
iInt := _w788;
_w13 := iInt + 1;
iInt := _w358;
iInt := _w359;
_w805 := iInt + 1;
iInt := _w526;
iInt := _w527;
iInt := _w589;
iInt := _w617;
iInt := _w636;
iInt := _w654;
iInt := _w672;
iInt := _w690;
iInt := _w708;
iInt := _w726;
iInt := _w805;
iInt := _w806;
_w807 := iInt + 1;
_w539 := iInt + 1;
_w540 := iInt + 1;
iInt := _w510;
iInt := _w546;
iInt := _w609;
iInt := _w628;
iInt := _w647;
iInt := _w665;
iInt := _w683;
iInt := _w701;
iInt := _w719;
iInt := _w191;
_w541 := iInt + 1;
_w542 := iInt + 1;
_w808 := iInt + 1;
_w809 := iInt + 1;
iInt := _w557;
iInt := _w612;
iInt := _w631;
iInt := _w649;
iInt := _w667;
iInt := _w685;
iInt := _w703;
iInt := _w721;
iInt := _w730;
iInt := _w809;
_w810 := iInt + 1;
iInt := _w584;
_w811 := iInt + 1;
iInt := _w585;
iInt := _w613;
iInt := _w632;
iInt := _w650;
iInt := _w668;
iInt := _w686;
iInt := _w704;
iInt := _w722;
iInt := _w731;
iInt := _w811;
iInt := _w470;
_w812 := iInt + 1;
iInt := _w751;
_w813 := iInt + 1;
iInt := _w734;
_w814 := iInt + 1;
_w815 := iInt + 1;
_w816 := iInt + 1;
_w817 := iInt + 1;
_w374 := iInt + 1;
_w401 := iInt + 1;
_w385 := iInt + 1;
_w818 := iInt + 1;
_w224 := iInt + 1;
_w736 := iInt + 1;
_w235 := iInt + 1;
_w602 := iInt + 1;
_w298 := iInt + 1;
_w603 := iInt + 1;
iInt := _w202;
_w604 := iInt + 1;
_w605 := iInt + 1;
_w819 := iInt + 1;
iInt := _w611;
iInt := _w630;
iInt := _w648;
iInt := _w666;
iInt := _w684;
iInt := _w702;
iInt := _w720;
iInt := _w729;
iInt := _w808;
iInt := _w121;
iInt := _w601;
iInt := _w620;
iInt := _w639;
iInt := _w657;
iInt := _w675;
iInt := _w693;
iInt := _w711;
iInt := _w122;
iInt := _w218;
iInt := _w819;
_w820 := iInt + 1;
_w821 := iInt + 1;
_w822 := iInt + 1;
_w823 := iInt + 1;
_w824 := iInt + 1;
_w825 := iInt + 1;
_w826 := iInt + 1;
_w827 := iInt + 1;
_w828 := iInt + 1;
_w556 := iInt + 1;
_w829 := iInt + 1;
_w830 := iInt + 1;
_w453 := iInt + 1;
_w831 := iInt + 1;
iInt := _w752;
iInt := _w753;
_w832 := iInt + 1;
iInt := _w770;
iInt := _w771;
_w833 := iInt + 1;
_w834 := iInt + 1;
iInt := _w789;
iInt := _w790;
_w375 := iInt + 1;
_w402 := iInt + 1;
_w386 := iInt + 1;
_w835 := iInt + 1;
iInt := _w30;
iInt := _w31;
_w225 := iInt + 1;
_w737 := iInt + 1;
_w236 := iInt + 1;
_w621 := iInt + 1;
_w299 := iInt + 1;
_w622 := iInt + 1;
iInt := _w203;
_w623 := iInt + 1;
_w624 := iInt + 1;
iInt := _w820;
_w836 := iInt + 1;
_w837 := iInt + 1;
_w454 := iInt + 1;
_w838 := iInt + 1;
iInt := _w754;
iInt := _w755;
_w839 := iInt + 1;
iInt := _w772;
iInt := _w773;
_w840 := iInt + 1;
_w841 := iInt + 1;
iInt := _w791;
iInt := _w792;
_w376 := iInt + 1;
_w403 := iInt + 1;
_w387 := iInt + 1;
_w842 := iInt + 1;
iInt := _w32;
iInt := _w33;
_w226 := iInt + 1;
_w738 := iInt + 1;
_w237 := iInt + 1;
_w640 := iInt + 1;
_w300 := iInt + 1;
_w641 := iInt + 1;
iInt := _w204;
_w642 := iInt + 1;
_w643 := iInt + 1;
iInt := _w821;
_w843 := iInt + 1;
_w844 := iInt + 1;
_w455 := iInt + 1;
_w845 := iInt + 1;
iInt := _w756;
iInt := _w757;
_w846 := iInt + 1;
iInt := _w774;
iInt := _w775;
_w847 := iInt + 1;
_w848 := iInt + 1;
iInt := _w793;
iInt := _w794;
_w377 := iInt + 1;
_w404 := iInt + 1;
_w388 := iInt + 1;
_w849 := iInt + 1;
iInt := _w34;
iInt := _w35;
_w227 := iInt + 1;
_w739 := iInt + 1;
_w238 := iInt + 1;
_w658 := iInt + 1;
_w301 := iInt + 1;
_w659 := iInt + 1;
iInt := _w205;
_w660 := iInt + 1;
_w661 := iInt + 1;
iInt := _w822;
_w850 := iInt + 1;
_w851 := iInt + 1;
_w456 := iInt + 1;
_w852 := iInt + 1;
iInt := _w758;
iInt := _w759;
_w853 := iInt + 1;
iInt := _w776;
iInt := _w777;
_w854 := iInt + 1;
_w855 := iInt + 1;
iInt := _w795;
iInt := _w796;
_w378 := iInt + 1;
_w405 := iInt + 1;
_w389 := iInt + 1;
_w856 := iInt + 1;
iInt := _w36;
iInt := _w37;
_w228 := iInt + 1;
_w740 := iInt + 1;
_w239 := iInt + 1;
_w676 := iInt + 1;
_w302 := iInt + 1;
_w677 := iInt + 1;
iInt := _w206;
_w678 := iInt + 1;
_w679 := iInt + 1;
iInt := _w823;
_w857 := iInt + 1;
_w858 := iInt + 1;
_w457 := iInt + 1;
_w859 := iInt + 1;
iInt := _w760;
iInt := _w761;
_w860 := iInt + 1;
iInt := _w778;
iInt := _w779;
_w861 := iInt + 1;
_w862 := iInt + 1;
iInt := _w797;
iInt := _w798;
_w379 := iInt + 1;
_w406 := iInt + 1;
_w390 := iInt + 1;
_w863 := iInt + 1;
iInt := _w38;
iInt := _w39;
_w229 := iInt + 1;
_w741 := iInt + 1;
_w240 := iInt + 1;
_w694 := iInt + 1;
_w303 := iInt + 1;
_w695 := iInt + 1;
iInt := _w207;
_w696 := iInt + 1;
_w697 := iInt + 1;
iInt := _w824;
_w864 := iInt + 1;
_w865 := iInt + 1;
_w458 := iInt + 1;
_w866 := iInt + 1;
iInt := _w762;
iInt := _w763;
_w867 := iInt + 1;
iInt := _w780;
iInt := _w781;
_w868 := iInt + 1;
_w869 := iInt + 1;
iInt := _w799;
iInt := _w800;
_w380 := iInt + 1;
_w407 := iInt + 1;
_w391 := iInt + 1;
_w870 := iInt + 1;
iInt := _w40;
iInt := _w41;
_w230 := iInt + 1;
_w742 := iInt + 1;
_w241 := iInt + 1;
_w712 := iInt + 1;
_w304 := iInt + 1;
_w713 := iInt + 1;
iInt := _w208;
_w714 := iInt + 1;
_w715 := iInt + 1;
iInt := _w825;
_w871 := iInt + 1;
_w872 := iInt + 1;
_w459 := iInt + 1;
_w873 := iInt + 1;
iInt := _w764;
iInt := _w765;
_w874 := iInt + 1;
iInt := _w782;
iInt := _w783;
_w875 := iInt + 1;
_w876 := iInt + 1;
iInt := _w801;
iInt := _w802;
_w381 := iInt + 1;
_w408 := iInt + 1;
_w392 := iInt + 1;
_w877 := iInt + 1;
iInt := _w42;
iInt := _w43;
_w231 := iInt + 1;
_w743 := iInt + 1;
_w242 := iInt + 1;
_w156 := iInt + 1;
_w305 := iInt + 1;
_w190 := iInt + 1;
iInt := _w209;
_w212 := iInt + 1;
_w214 := iInt + 1;
iInt := _w826;
_w878 := iInt + 1;
_w879 := iInt + 1;
_w460 := iInt + 1;
_w880 := iInt + 1;
iInt := _w766;
iInt := _w767;
_w881 := iInt + 1;
iInt := _w784;
iInt := _w785;
_w882 := iInt + 1;
_w883 := iInt + 1;
iInt := _w803;
iInt := _w804;
_w382 := iInt + 1;
_w409 := iInt + 1;
_w393 := iInt + 1;
_w884 := iInt + 1;
iInt := _w807;
iInt := _w818;
iInt := _w835;
iInt := _w842;
iInt := _w849;
iInt := _w856;
iInt := _w863;
iInt := _w870;
iInt := _w877;
iInt := _w884;
_w397 := iInt + 1;
_w399 := iInt + 1;
iInt := _w827;
_w885 := iInt + 1;
_w886 := iInt + 1;
_w461 := iInt + 1;
_w887 := iInt + 1;
iInt := _w812;
iInt := _w831;
iInt := _w838;
iInt := _w845;
iInt := _w852;
iInt := _w859;
iInt := _w866;
iInt := _w873;
iInt := _w880;
iInt := _w887;
_w167 := iInt + 1;
iInt := _w768;
iInt := _w769;
_w888 := iInt + 1;
iInt := _w813;
_w889 := iInt + 1;
_w890 := iInt + 1;
_w891 := iInt + 1;
_w892 := iInt + 1;
_w893 := iInt + 1;
_w894 := iInt + 1;
_w895 := iInt + 1;
_w896 := iInt + 1;
_w897 := iInt + 1;
_w898 := iInt + 1;
_w899 := iInt + 1;
_w900 := iInt + 1;
_w901 := iInt + 1;
_w902 := iInt + 1;
_w903 := iInt + 1;
_w904 := iInt + 1;
_w78 := iInt + 1;
_w79 := iInt + 1;
iInt := _w814;
iInt := _w832;
iInt := _w839;
iInt := _w846;
iInt := _w853;
iInt := _w860;
iInt := _w867;
iInt := _w874;
iInt := _w881;
iInt := _w888;
_w111 := iInt + 1;
iInt := _w786;
iInt := _w787;
_w905 := iInt + 1;
iInt := _w815;
iInt := _w816;
iInt := _w833;
iInt := _w840;
iInt := _w847;
iInt := _w854;
iInt := _w861;
iInt := _w868;
iInt := _w875;
iInt := _w882;
iInt := _w905;
iInt := _w142;
_w906 := iInt + 1;
_w543 := iInt + 1;
iInt := _w528;
iInt := _w590;
iInt := _w618;
iInt := _w637;
iInt := _w655;
iInt := _w673;
iInt := _w691;
iInt := _w709;
iInt := _w727;
iInt := _w907;
_w544 := iInt + 1;
_w545 := iInt + 1;
iInt := _w828;
_w908 := iInt + 1;
iInt := _w829;
iInt := _w836;
iInt := _w843;
iInt := _w850;
iInt := _w857;
iInt := _w864;
iInt := _w871;
iInt := _w878;
iInt := _w885;
iInt := _w908;
iInt := _w909;
_w910 := iInt + 1;
iInt := _w586;
iInt := _w614;
iInt := _w633;
iInt := _w651;
iInt := _w669;
iInt := _w687;
iInt := _w705;
iInt := _w723;
iInt := _w732;
iInt := _w452;
_w472 := iInt + 1;
_w529 := iInt + 1;
_w81 := iInt + 1;
_w592 := iInt + 1;
_w125 := iInt + 1;
_w911 := iInt + 1;
_w4 := iInt + 1;
_w606 := iInt + 1;
iInt := _w912;
_w607 := iInt + 1;
_w608 := iInt + 1;
_w913 := iInt + 1;
_w914 := iInt + 1;
iInt := _w462;
_w473 := iInt + 1;
_w530 := iInt + 1;
iInt := _w889;
iInt := _w890;
_w82 := iInt + 1;
_w593 := iInt + 1;
_w126 := iInt + 1;
_w915 := iInt + 1;
_w5 := iInt + 1;
_w625 := iInt + 1;
iInt := _w916;
_w626 := iInt + 1;
_w627 := iInt + 1;
_w917 := iInt + 1;
_w918 := iInt + 1;
iInt := _w463;
_w474 := iInt + 1;
_w531 := iInt + 1;
iInt := _w891;
iInt := _w892;
_w83 := iInt + 1;
_w594 := iInt + 1;
_w127 := iInt + 1;
_w919 := iInt + 1;
_w6 := iInt + 1;
_w644 := iInt + 1;
iInt := _w920;
_w645 := iInt + 1;
_w646 := iInt + 1;
_w921 := iInt + 1;
_w922 := iInt + 1;
iInt := _w464;
_w475 := iInt + 1;
_w532 := iInt + 1;
iInt := _w893;
iInt := _w894;
_w84 := iInt + 1;
_w595 := iInt + 1;
_w128 := iInt + 1;
_w923 := iInt + 1;
_w7 := iInt + 1;
_w662 := iInt + 1;
iInt := _w924;
_w663 := iInt + 1;
_w664 := iInt + 1;
_w925 := iInt + 1;
_w926 := iInt + 1;
iInt := _w465;
_w476 := iInt + 1;
_w533 := iInt + 1;
iInt := _w895;
iInt := _w896;
_w85 := iInt + 1;
_w596 := iInt + 1;
_w129 := iInt + 1;
_w927 := iInt + 1;
_w8 := iInt + 1;
_w680 := iInt + 1;
iInt := _w928;
_w681 := iInt + 1;
_w682 := iInt + 1;
_w929 := iInt + 1;
_w930 := iInt + 1;
iInt := _w466;
_w477 := iInt + 1;
_w534 := iInt + 1;
iInt := _w897;
iInt := _w898;
_w86 := iInt + 1;
_w597 := iInt + 1;
_w130 := iInt + 1;
_w931 := iInt + 1;
_w9 := iInt + 1;
_w698 := iInt + 1;
iInt := _w932;
_w699 := iInt + 1;
_w700 := iInt + 1;
_w933 := iInt + 1;
_w934 := iInt + 1;
iInt := _w467;
_w478 := iInt + 1;
_w535 := iInt + 1;
iInt := _w899;
iInt := _w900;
_w87 := iInt + 1;
_w598 := iInt + 1;
_w131 := iInt + 1;
_w935 := iInt + 1;
_w10 := iInt + 1;
_w716 := iInt + 1;
iInt := _w936;
_w717 := iInt + 1;
_w718 := iInt + 1;
_w937 := iInt + 1;
_w938 := iInt + 1;
iInt := _w468;
_w479 := iInt + 1;
_w536 := iInt + 1;
iInt := _w901;
iInt := _w902;
_w88 := iInt + 1;
_w599 := iInt + 1;
_w132 := iInt + 1;
_w939 := iInt + 1;
_w11 := iInt + 1;
_w384 := iInt + 1;
iInt := _w940;
_w396 := iInt + 1;
_w398 := iInt + 1;
_w941 := iInt + 1;
_w942 := iInt + 1;
iInt := _w469;
_w480 := iInt + 1;
_w537 := iInt + 1;
iInt := _w903;
iInt := _w904;
_w89 := iInt + 1;
_w600 := iInt + 1;
_w133 := iInt + 1;
_w943 := iInt + 1;
iInt := _w906;
iInt := _w911;
iInt := _w915;
iInt := _w919;
iInt := _w923;
iInt := _w927;
iInt := _w931;
iInt := _w935;
iInt := _w939;
iInt := _w943;
_w566 := iInt + 1;
_w93 := iInt + 1;
iInt := _w817;
iInt := _w834;
iInt := _w841;
iInt := _w848;
iInt := _w855;
iInt := _w862;
iInt := _w869;
iInt := _w876;
iInt := _w883;
iInt := _w124;
_w144 := iInt + 1;
_w567 := iInt + 1;
_w103 := iInt + 1;
_w94 := iInt + 1;
iInt := _w134;
_w145 := iInt + 1;
_w568 := iInt + 1;
_w104 := iInt + 1;
_w95 := iInt + 1;
iInt := _w135;
_w146 := iInt + 1;
_w569 := iInt + 1;
_w105 := iInt + 1;
_w96 := iInt + 1;
iInt := _w136;
_w147 := iInt + 1;
_w570 := iInt + 1;
_w106 := iInt + 1;
_w97 := iInt + 1;
iInt := _w137;
_w148 := iInt + 1;
_w571 := iInt + 1;
_w107 := iInt + 1;
_w98 := iInt + 1;
iInt := _w138;
_w149 := iInt + 1;
_w572 := iInt + 1;
_w108 := iInt + 1;
_w99 := iInt + 1;
iInt := _w139;
_w150 := iInt + 1;
_w573 := iInt + 1;
_w109 := iInt + 1;
_w100 := iInt + 1;
iInt := _w140;
_w151 := iInt + 1;
_w574 := iInt + 1;
_w110 := iInt + 1;
_w101 := iInt + 1;
iInt := _w141;
_w152 := iInt + 1;
_w575 := iInt + 1;
_w944 := iInt + 1;
_w945 := iInt + 1;
iInt := _w910;
iInt := _w914;
iInt := _w918;
iInt := _w922;
iInt := _w926;
iInt := _w930;
iInt := _w934;
iInt := _w938;
iInt := _w942;
iInt := _w945;
_w946 := iInt + 1;
_w947 := iInt + 1;
iInt := _w913;
iInt := _w917;
iInt := _w921;
iInt := _w925;
iInt := _w929;
iInt := _w933;
iInt := _w937;
iInt := _w941;
iInt := _w944;
iInt := _w810;
iInt := _w830;
iInt := _w837;
iInt := _w844;
iInt := _w851;
iInt := _w858;
iInt := _w865;
iInt := _w872;
iInt := _w879;
iInt := _w886;
iInt := _w947;
_w948 := iInt + 1;
_w949 := iInt + 1;
_w950 := iInt + 1;
_w951 := iInt + 1;
_w952 := iInt + 1;
_w953 := iInt + 1;
_w954 := iInt + 1;
_w955 := iInt + 1;
_w909 := iInt + 1;
_w956 := iInt + 1;
_w957 := iInt + 1;
iInt := iInt + 1;
_w958 := iInt + 1;
_w959 := iInt + 1;
iInt := _w948;
_w960 := iInt + 1;
_w961 := iInt + 1;
iInt := _w949;
_w962 := iInt + 1;
_w963 := iInt + 1;
iInt := _w950;
_w964 := iInt + 1;
_w965 := iInt + 1;
iInt := _w951;
_w966 := iInt + 1;
_w967 := iInt + 1;
iInt := _w952;
_w968 := iInt + 1;
_w969 := iInt + 1;
iInt := _w953;
_w970 := iInt + 1;
_w971 := iInt + 1;
iInt := _w954;
_w972 := iInt + 1;
_w973 := iInt + 1;
iInt := _w211;
iInt := _w955;
_w974 := iInt + 1;
iInt := _w956;
iInt := _w958;
iInt := _w960;
iInt := _w962;
iInt := _w964;
iInt := _w966;
iInt := _w968;
iInt := _w970;
iInt := _w972;
iInt := _w974;
_w975 := iInt + 1;
_w976 := iInt + 1;
_w977 := iInt + 1;
_w978 := iInt + 1;
_w979 := iInt + 1;
_w980 := iInt + 1;
_w981 := iInt + 1;
_w982 := iInt + 1;
_w907 := iInt + 1;
_w912 := iInt + 1;
_w916 := iInt + 1;
_w920 := iInt + 1;
_w924 := iInt + 1;
_w928 := iInt + 1;
_w932 := iInt + 1;
_w936 := iInt + 1;
_w940 := iInt + 1;
_w394 := iInt + 1;
_w806 := iInt + 1;
_w983 := iInt + 1;
iInt := iInt + 1;
iInt := _w975;
iInt := _w976;
iInt := _w977;
iInt := _w978;
iInt := _w979;
iInt := _w980;
iInt := _w981;
iInt := _w982;
iInt := _w946;
iInt := _w957;
iInt := _w959;
iInt := _w961;
iInt := _w963;
iInt := _w965;
iInt := _w967;
iInt := _w969;
iInt := _w971;
iInt := _w973;
iInt := _w983;

END_PROGRAM

// Device/Application/UserPOUs/Redundant/Languages/POU_FBD
PROGRAM POU_FBD
VAR
	/// Variáveis para testar ADD de 2 entradas
	bHab01: BOOL := FALSE;
	iSom01A: INT := 1;
	iSom01B: INT := 2;
	/// valor esperado = 3
	iSom01R: INT;
	/// Variáveis para testar ADD de 3 entradas
	bHab02: BOOL := TRUE;
	iSom02A: INT := 1;
	iSom02B: INT := 2;
	iSom02C: INT := 3;
	/// valor esperado = 6
	iSom02R: INT;
	/// Variáveis para testar SUB de 2 entradas
	bHab03: BOOL := TRUE;
	iSub03A: INT := 3;
	iSub03B: INT := 2;
	/// valor esperado = 1
	iSub03R: INT;
	/// Variáveis para testar MUL de 2 entradas
	bHab04: BOOL := TRUE;
	iMul04A: INT := 4;
	iMul04B: INT := 4;
	/// valor esperado = 16
	iMul04R: INT;
	/// Variáveis para testar DIV de 2 entradas
	bHab05: BOOL := TRUE;
	iDiv05A: INT := 20;
	iDiv05B: INT := 5;
	/// valor esperado = 4
	iDiv05R: INT;
	/// Variáveis para testar EQ de 2 entradas
	bHab06: BOOL := FALSE;
	iEq06A: INT := 25;
	iEq06B: INT := 25;
	/// valor esperado = true	
	bEq06R: BOOL;
	/// Variáveis para testar NE de 2 entradas
	bHab07: BOOL := TRUE;
	iNe07A: INT := 24;
	iNe07B: INT := 25;
	/// valor esperado = true
	bNe07R: BOOL;
	/// Variáveis para testar LT de 2 entradas
	bHab08: BOOL := TRUE;
	iLt08A: INT := 24;
	iLt08B: INT := 25;
	/// valor esperado = true		
	bLt08R: BOOL;
	/// Variáveis para testar LE de 2 entradas
	bHab09: BOOL := TRUE;
	iLe09A: INT := 25;
	iLe09B: INT := 25;
	/// valor esperado = true		
	bLe09R: BOOL;
	/// Variáveis para testar GT de 2 entradas
	bHab10: BOOL := TRUE;
	iGt10A: INT := 26;
	iGt10B: INT := 25;
	/// valor esperado = true	
	bGt10R: BOOL;
	/// Variáveis para testar GE de 2 entradas
	bHab11: BOOL := TRUE;
	iGe11A: INT := 26;
	iGe11B: INT := 26;
	/// valor esperado = true		
	bGe11R: BOOL;
	/// Variáveis para testar SEL
	bHab12: BOOL := TRUE;
	bSelG: BOOL := TRUE;
	iSel12A: INT := 20;
	iSel12B: INT := 26;
	/// valor esperado = 26		
	iSel12R: INT;
	/// Variáveis para testar MUX
	bHab13: BOOL := TRUE;
	iMux13K: INT := 2;
	/// valor esperado = 30		
	iMux13R: INT;
	/// Variáveis para testar LIMIT
	bHab14: BOOL := TRUE;
	iLim14In: INT := 5;
	/// valor esperado = 20		
	iLim14R: INT;
	/// Variáveis para testar MOVE
	bHab15: BOOL := TRUE;
	iMov15In: INT := 5;
	/// valor esperado = 5
	iMov15R: INT;
	/// Variáveis para testar Conversão
	bHab16: BOOL := TRUE;
	/// valor esperado = 1	
	iConv16R: INT;
	/// Variáveis para testar elementos Ladder
	bContato01: BOOL := TRUE;
	/// valor esperado = 1	
	bContato01R: BOOL;
	bContato02: BOOL := FALSE;
	/// valor esperado = 1	
	bContato02R: BOOL;
	bContato03: BOOL := TRUE;
	/// valor esperado = 1	
	bContato03R: BOOL;
END_VAR

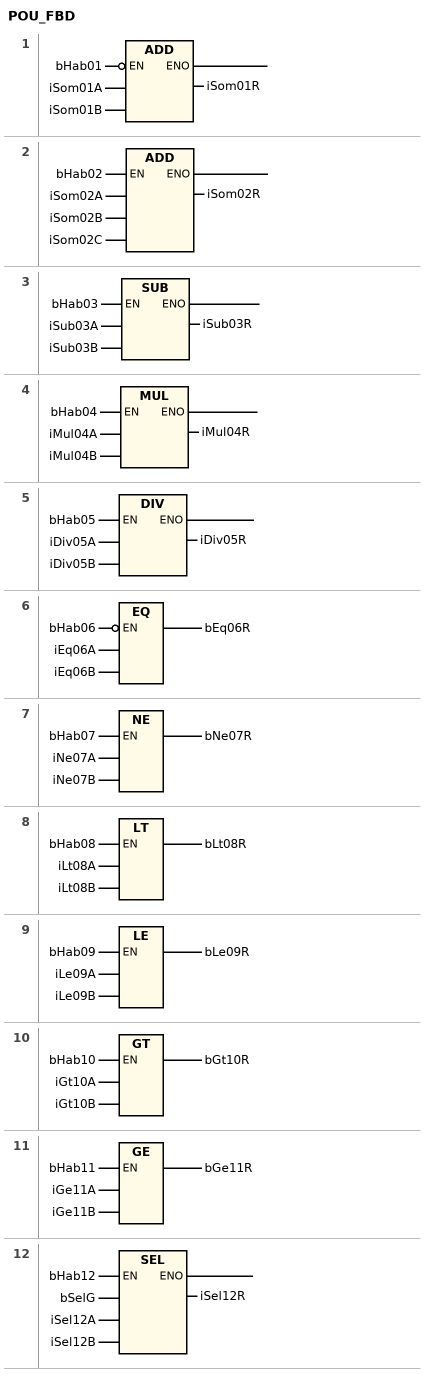
// NETWORK 1
IF NOT bHab01 THEN iSom01R := iSom01A + iSom01B; END_IF

// NETWORK 2
IF bHab02 THEN iSom02R := iSom02A + iSom02B + iSom02C; END_IF

// NETWORK 3
IF bHab03 THEN iSub03R := iSub03A - iSub03B; END_IF

// NETWORK 4
IF bHab04 THEN iMul04R := iMul04A * iMul04B; END_IF

// NETWORK 5
IF bHab05 THEN iDiv05R := iDiv05A / iDiv05B; END_IF

// NETWORK 6
bEq06R := NOT bHab06 AND iEq06A = iEq06B;

// NETWORK 7
bNe07R := bHab07 AND iNe07A <> iNe07B;

// NETWORK 8
bLt08R := bHab08 AND iLt08A < iLt08B;

// NETWORK 9
bLe09R := bHab09 AND iLe09A <= iLe09B;

// NETWORK 10
bGt10R := bHab10 AND iGt10A > iGt10B;

// NETWORK 11
bGe11R := bHab11 AND iGe11A >= iGe11B;

// NETWORK 12
IF bHab12 THEN iSel12R := SEL(bSelG, iSel12A, iSel12B); END_IF

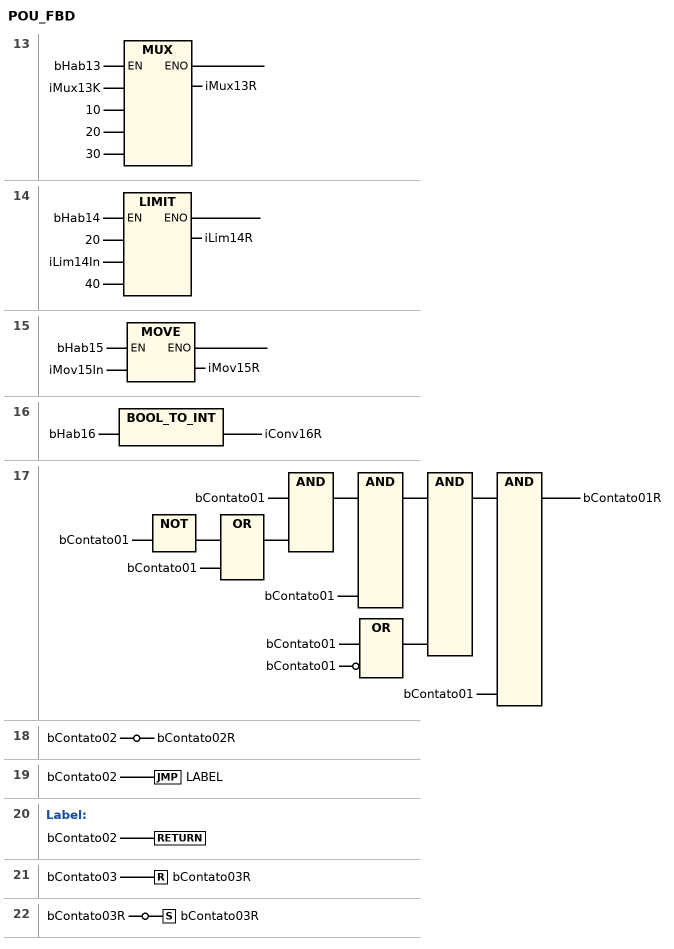
// NETWORK 13
IF bHab13 THEN iMux13R := MUX(iMux13K, 10, 20, 30); END_IF

// NETWORK 14
IF bHab14 THEN iLim14R := LIMIT(20, iLim14In, 40); END_IF

// NETWORK 15
IF bHab15 THEN iMov15R := iMov15In; END_IF

// NETWORK 16
iConv16R := BOOL_TO_INT(bHab16);

// NETWORK 17
bContato01R := (((bContato01 AND (NOT bContato01 OR bContato01)) AND bContato01) AND (bContato01 OR NOT bContato01)) AND bContato01;

// NETWORK 18
bContato02R := NOT bContato02;

// NETWORK 19
IF bContato02 THEN JMP LABEL; END_IF

// NETWORK 20
Label:
IF bContato02 THEN RETURN; END_IF

// NETWORK 21
bContato03R R= bContato03;

// NETWORK 22
bContato03R S= NOT bContato03R;

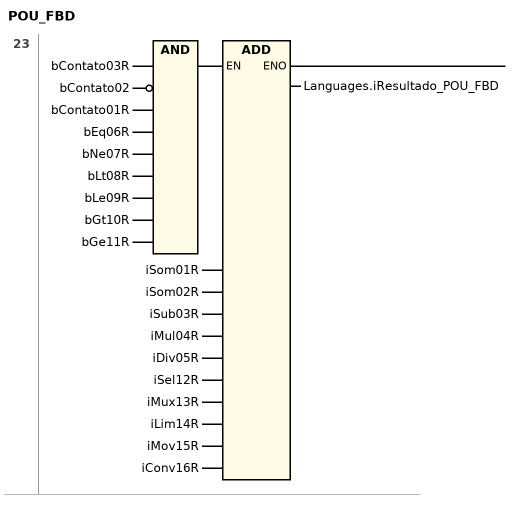
// NETWORK 23
IF bContato03R AND NOT bContato02 AND bContato01R AND bEq06R AND bNe07R AND bLt08R AND bLe09R AND bGt10R AND bGe11R THEN
    Languages.iResultado_POU_FBD := iSom01R + iSom02R + iSub03R + iMul04R + iDiv05R + iSel12R + iMux13R + iLim14R + iMov15R + iConv16R;
END_IF

END_PROGRAM

// Device/Application/UserPOUs/Redundant/Alarms
PROGRAM Alarms
VAR
	// UserLog para salvar no cartão o tempo que ocorreu o problema
	eLogError : liblogs.USER_LOG_ERROR_CODES;
	// USER_LOG_MESSAGE;
	sMessage : STRING(150);
	// Registra apenas o primeiro erro
	bOneCycle : BOOL := FALSE;
	uliPouIniTime : ULINT;
	uliPouEndTime : ULINT;
END_VAR

// Detecção dos alarmes mapeados no sistema de supervisão

// Registra o tempo do sistema
SysTimeGetUs(uliPouIniTime);

// Resumo do diagnóstico do PLC A e PLC B estão na GVL DiagRetain

// Forcing
PersistentVars.bForcing:=	PersistentVars.bForcingDiagUnset OR
							PersistentVars.bBoolVarNotForced OR
							PersistentVars.bWordVarNotForced;

// Languages
PersistentVars.bLanguages:= Persistentvars.dwErrorLanguages <> 0;	

// MODBUS_Master_1
PersistentVars.bModbus1:=	PersistentVars.bModbus1ErrorCoil OR
							PersistentVars.bModbus1ErrorStatus OR 
							PersistentVars.bModbus1ErrorHolding OR
							PersistentVars.bModbus1ErrorInputReg;
// MODBUS_Client_2
PersistentVars.bModbus2:=	PersistentVars.bModbus2ErrorCoil OR
							PersistentVars.bModbus2ErrorStatus OR 
							PersistentVars.bModbus2ErrorHolding OR
							PersistentVars.bModbus2ErrorInputReg;
// MODBUS_Client_3
PersistentVars.bModbus3:=	PersistentVars.bModbus3ErrorCoil OR
							PersistentVars.bModbus3ErrorStatus OR 
							PersistentVars.bModbus3ErrorHolding OR
							PersistentVars.bModbus3ErrorInputReg;
// MODBUS_Client_4
PersistentVars.bModbus4:=	PersistentVars.bModbus4ErrorCoil OR
							PersistentVars.bModbus4ErrorStatus OR
							PersistentVars.bModbus4ErrorHolding OR
							PersistentVars.bModbus4ErrorInputReg;

// Profibus
PersistentVars.bProfibusIOs:= 	PersistentVars.dwSlave5DigIOsErrors<>0 AND Mask.bug23167 OR
								PersistentVars.dwSlave5Unavailable<>0 OR
								PersistentVars.dwSlave5ModulesOut<>0 OR
								PersistentVars.dwSlave10AnaIOsErrors<>0 OR
								PersistentVars.dwSlave10Unavailable<>0 OR
								PersistentVars.dwSlave10ModulesOut<>0 OR
								PersistentVars.dwSlave3DigIOsErrors<>0 AND Mask.bug23167 OR
								PersistentVars.dwSlave3Unavailable<>0 OR
								PersistentVars.dwSlave3ModulesOut <>0 OR
								//Gabriel Fonseca - 28/10/2022
								//Alterado para tornar toleravel no maximo 1 erro por hora
								//Torna toleravel um erro por hora
								PersistentVars.dwSlave5DigIOsErrors > (TIME_TO_DWORD (PersistentVars.tElapsedTimeToFailure)/3600000) + 1 OR  
								PersistentVars.dwSlave3DigIOsErrors > (TIME_TO_DWORD (PersistentVars.tElapsedTimeToFailure)/3600000) + 1 OR
								//Indica falha caso congele por mais de um ciclo 
								PersistentVars.bFrozenErrorRem05TORem05 OR 
								PersistentVars.bFrozenErrorRem05TORem04;
								

/// Recipe Manager
PersistentVars.bRecipeManager:= Persistentvars.dwRecipeErrors <> 0 OR
							    Persistentvars.dwRecipeReturnError <> 0;

// Redundant Data
PersistentVars.bRedundantData:= PersistentVars.iSyncFailCntSymb <> 0 OR
								PersistentVars.iSyncFailCntQ <> 0 OR
								PersistentVars.iSyncFailCntM <> 0 OR
								PersistentVars.iSyncFailCntI <> 0 OR
								PersistentVars.iSyncFailCallback_vfInit <> 0;

// Redundant state
PersistentVars.bRedundantState:= PersistentVars.bExchangeStateFail;

// SNTP
PersistentVars.bSntp:=	PersistentVars.bSntpSourceFailures OR
						PersistentVars.bSntpServerFailures OR
						PersistentVars.bTimezoneFailure OR
						PersistentVars.iSntpSyncFailures > 0;

// SOE
PersistentVars.bSOE:=	PersistentVars.bSOE1EventsMismatch OR
						PersistentVars.bSOE1FalseOverflow OR
						PersistentVars.bSOE2EventsMismatch OR
						PersistentVars.bSOE2FalseOverflow;

// Ram
PersistentVars.bRam:=	PersistentVars.bRamTotalFailure OR
						PersistentVars.bRamFreeVarFailure;
						
// Detecção de falha geral
PersistentVars.bFailureDetected:=	PersistentVars.bActiveDiagPlcA OR
									PersistentVars.bActiveDiagPlcB OR
									PersistentVars.bForcing OR
									PersistentVars.bLanguages OR
									PersistentVars.bModbus1 OR
									PersistentVars.bModbus2 OR
									PersistentVars.bModbus3 OR
									PersistentVars.bModbus4 OR
									PersistentVars.bProfibusIOs OR
									PersistentVars.bRecipeManager OR
									PersistentVars.bRedundantData OR
									PersistentVars.bRedundantState OR
									PersistentVars.bSNTP OR
									PersistentVars.bSOE OR
									PersistentVars.bSpecialVariables OR
									PersistentVars.bUserLog OR
									PersistentVars.bRam OR
									StartPrg.bCheckAppGetInfo;



IF 	PersistentVars.bFailureDetected THEN								
	// Liga LED para indicar um erro visual
	REM10_PO2132_C03:= 30000;
	// Resgitra o momento que ocorreu o problema.
	IF bOneCycle = FALSE THEN
		sMessage := ' Instante:; ';
		sMessage := concat(sMessage, TIME_TO_STRING(PersistentVars.tElapsedTimeToFailure));
		sMessage := concat(sMessage,' ;Resultado:; NOK');
		eLogError := UserLogAdd(USER_LOG_EVENT_ERROR, sMessage);
		bOneCycle:= TRUE;
	END_IF	
ELSE
	// Desliga LED para indicar que não há erro de forma visual
	REM10_PO2132_C03:= 00;
	bOneCycle:= FALSE;
END_IF

// Registra o tempo do sistema
SysTimeGetUs(uliPouEndTime);
// Calcula duração mínima/máxima desta POU
MinMaxTimes.uliPouMinTime_Alarms:= MIN(MinMaxTimes.uliPouMinTime_Alarms, uliPouEndTime - uliPouIniTime);
MinMaxTimes.uliPouMaxTime_Alarms:= MAX(MinMaxTimes.uliPouMaxTime_Alarms, uliPouEndTime - uliPouIniTime);

END_PROGRAM

// Device/Application/UserPOUs/Non-Redundant/UserLog
PROGRAM UserLog
VAR
	// UserLog
	eLogError : liblogs.USER_LOG_ERROR_CODES;
	// UserLog message
	sMessage : STRING(150);
	uliPouIniTime : ULINT;
	uliPouEndTime : ULINT;
END_VAR

// Testa a funcionalidade do LOG de usuário

// Registra o tempo do sistema
SysTimeGetUs(uliPouIniTime);

// Ao iniciar o teste, registra no UserLog a data e hora de inicio
IF Symbolics.bStartTestCopy = TRUE THEN
	IF NonRedData.iStepUserlog = 2 THEN	
		sMessage := ' Inicio teste:; ';
	 	sMessage := concat(sMessage, WORD_TO_STRING(NonRedData.xNonSkippedPrgDateAndTime.wYear));
		sMessage := concat(sMessage,'-');
		sMessage := concat(sMessage, BYTE_TO_STRING(NonRedData.xNonSkippedPrgDateAndTime.byMonth));
		sMessage := concat(sMessage,'-');
		sMessage := concat(sMessage, BYTE_TO_STRING(NonRedData.xNonSkippedPrgDateAndTime.byDayOfMonth));
		sMessage := concat(sMessage,'-');
		sMessage := concat(sMessage, BYTE_TO_STRING(NonRedData.xNonSkippedPrgDateAndTime.byHours));
		sMessage := concat(sMessage,':');
		sMessage := concat(sMessage, BYTE_TO_STRING(NonRedData.xNonSkippedPrgDateAndTime.byMinutes));
		sMessage := concat(sMessage,':');
		sMessage := concat(sMessage, BYTE_TO_STRING(NonRedData.xNonSkippedPrgDateAndTime.bySeconds));
		sMessage := concat(sMessage,':');
		sMessage := concat(sMessage, WORD_TO_STRING(NonRedData.xNonSkippedPrgDateAndTime.wMilliseconds));
		sMessage := concat(sMessage,' ;Resultado:; Pendente');
		eLogError := UserLogAdd(USER_LOG_EVENT_INFO, sMessage);	
		NonRedData.iStepUserlog := 3;
	END_IF
	IF NonRedData.iStepUserlog < 2 THEN // Defasa o registro em dois ciclos para atualizar o relógio da UCP.
		NonRedData.iStepUserlog := NonRedData.iStepUserlog+1;
	END_IF
END_IF

// Ao completar 2 dias sem nenhum erro, registra no UserLog a data e hora do fim
IF (PersistentVars.tElapsedTimeToFailure > NonRedData.tMinimumTime AND PersistentVars.bFailureDetected = FALSE)  THEN
	IF NonRedData.iStepUserlog = 3 THEN	
		sMessage := 'Fim teste:; ';
		sMessage := concat(sMessage, WORD_TO_STRING(NonRedData.xNonSkippedPrgDateAndTime.wYear));
		sMessage := concat(sMessage,'/');
		sMessage := concat(sMessage, BYTE_TO_STRING(NonRedData.xNonSkippedPrgDateAndTime.byMonth));
		sMessage := concat(sMessage,'/');
		sMessage := concat(sMessage, BYTE_TO_STRING(NonRedData.xNonSkippedPrgDateAndTime.byDayOfMonth));
		sMessage := concat(sMessage,' ');
		sMessage := concat(sMessage, BYTE_TO_STRING(NonRedData.xNonSkippedPrgDateAndTime.byHours));
		sMessage := concat(sMessage,':');
		sMessage := concat(sMessage, BYTE_TO_STRING(NonRedData.xNonSkippedPrgDateAndTime.byMinutes));
		sMessage := concat(sMessage,':');
		sMessage := concat(sMessage, BYTE_TO_STRING(NonRedData.xNonSkippedPrgDateAndTime.bySeconds));
		sMessage := concat(sMessage,'.');
		sMessage := concat(sMessage, WORD_TO_STRING(NonRedData.xNonSkippedPrgDateAndTime.wMilliseconds));
		sMessage := concat(sMessage,' ;CRC da Aplicação:; ');
		sMessage := concat(sMessage, DWORD_TO_STRING(DG_NX3030.tDetailed.ApplicationInfo.dwApplicationCRC));
		sMessage := concat(sMessage,' ;Resultado:; Aprovado');
		sMessage := concat(sMessage,' ;TC Mín A:; ');
		sMessage := concat(sMessage, DWORD_TO_STRING(PersistentVars.dwPLCAMainTaskMinScanTime));
		sMessage := concat(sMessage,' ;TC Méd A:; ');
		sMessage := concat(sMessage, DWORD_TO_STRING(PersistentVars.dwPLCAMainTaskAvgScanTime));
		sMessage := concat(sMessage,' ;TC Máx A:; ');
		sMessage := concat(sMessage, DWORD_TO_STRING(PersistentVars.dwPLCAMainTaskMaxScanTime));
		eLogError := UserLogAdd(USER_LOG_EVENT_INFO, sMessage);	
		NonRedData.iStepUserlog := 4;
	END_IF
END_IF

 // Gera erro, caso a função do UserLog retorne algum erro.
IF eLogError <> 0 THEN
	NonRedPointer.pbErrorUserLogLoc^ := TRUE;
	Persistentvars.bUserLog:= 	NonRedPointer.pbErrorUserLogLoc^ OR
								NonRedPointer.pbErrorUserLogRem^;
END_IF

// Registra o tempo do sistema
SysTimeGetUs(uliPouEndTime);
// Calcula duração mínima/máxima desta POU
MinMaxTimes.uliPouMinTime_UserLog:= MIN(MinMaxTimes.uliPouMinTime_UserLog, uliPouEndTime - uliPouIniTime);
MinMaxTimes.uliPouMaxTime_UserLog:= MAX(MinMaxTimes.uliPouMaxTime_UserLog, uliPouEndTime - uliPouIniTime);

END_PROGRAM

// Device/Application/UserPOUs/Redundant/CheckNVL
PROGRAM CheckNVL
VAR
	// Quantidade de ciclos sem comunicação com a JIGA01
	iJIGA01_CiclosSemComunicao : INT;
	// Quantidade de ciclos sem comunicação com a JIGA02
	iJIGA02_CiclosSemComunicao : INT;
	// Quantidade de ciclos sem comunicação com a JIGA03
	iJIGA03_CiclosSemComunicao : INT;
	// Quantidade de ciclos sem comunicação com a JIGA05
	iJIGA05_CiclosSemComunicao : INT;
	// Quantidade de ciclos sem comunicação com a JIGA07
	iJIGA07_CiclosSemComunicao : INT;
	// Quantidade máxima de ciclos sem comunicação com a JIGA01
	iJIGA01_CiclosSemComunicaoMax : INT;
	// Quantidade máxima de ciclos sem comunicação com a JIGA02
	iJIGA02_CiclosSemComunicaoMax : INT;
	// Quantidade máxima de ciclos sem comunicação com a JIGA03
	iJIGA03_CiclosSemComunicaoMax : INT;
	// Quantidade máxima de ciclos sem comunicação com a JIGA05 
	iJIGA05_CiclosSemComunicaoMax : INT;
	// Quantidade máxima de ciclos sem comunicação com a JIGA07 
	iJIGA07_CiclosSemComunicaoMax : INT;
	// Contador de comunicações que houveram com a JIGA01
	ctuJIGA01_QtdComunicao : CTU;
	// Contador de comunicações que houveram com a JIGA02
	ctuJIGA02_QtdComunicao : CTU;
	// Contador de comunicações que houveram com a JIGA03
	ctuJIGA03_QtdComunicao : CTU;
	// Contador de comunicações que houveram com a JIGA05
	ctuJIGA05_QtdComunicao : CTU;
	// Contador de comunicações que houveram com a JIGA07
	ctuJIGA07_QtdComunicao : CTU;
	// Contador de comunicações que demoraram mais de 3 segundos com a JIGA01
	ctuJIGA01_QtdComunicao3s : CTU;
	// Contador de comunicações que demoraram mais de 3 segundos com a JIGA02
	ctuJIGA02_QtdComunicao3s : CTU;
	// Contador de comunicações que demoraram mais de 3 segundos com a JIGA03
	ctuJIGA03_QtdComunicao3s : CTU;
	// Contador de comunicações que demoraram mais de 3 segundos com a JIGA05
	ctuJIGA05_QtdComunicao3s : CTU;
	// Contador de comunicações que demoraram mais de 3 segundos com a JIGA07
	ctuJIGA07_QtdComunicao3s : CTU;
	// Contador de comunicações que demoraram mais de 4 segundos com a JIGA01
	ctuJIGA01_QtdComunicao4s : CTU;
	// Contador de comunicações que demoraram mais de 4 segundos com a JIGA02
	ctuJIGA02_QtdComunicao4s : CTU;
	// Contador de comunicações que demoraram mais de 4 segundos com a JIGA03
	ctuJIGA03_QtdComunicao4s : CTU;
	// Contador de comunicações que demoraram mais de 4 segundos com a JIGA05
	ctuJIGA05_QtdComunicao4s : CTU;
	// Contador de comunicações que demoraram mais de 4 segundos com a JIGA07
	ctuJIGA07_QtdComunicao4s : CTU;
	// Contador de comunicações que demoraram mais de 5 segundos com a JIGA01
	ctuJIGA01_QtdComunicao5s : CTU;
	// Contador de comunicações que demoraram mais de 5 segundos com a JIGA02
	ctuJIGA02_QtdComunicao5s : CTU;
	// Contador de comunicações que demoraram mais de 5 segundos com a JIGA03
	ctuJIGA03_QtdComunicao5s : CTU;
	// Contador de comunicações que demoraram mais de 5 segundos com a JIGA05
	ctuJIGA05_QtdComunicao5s : CTU;
	// Contador de comunicações que demoraram mais de 5 segundos com a JIGA07
	ctuJIGA07_QtdComunicao5s : CTU;
	// Estatísticas de comunicações com a JIGA01
	statJIGA01_Comunicacao : statistics_int;
	// Estatísticas de comunicações com a JIGA02
	statJIGA02_Comunicacao : statistics_int;
	// Estatísticas de comunicações com a JIGA03
	statJIGA03_Comunicacao : statistics_int;
	// Estatísticas de comunicações com a JIGA05
	statJIGA05_Comunicacao : statistics_int;
	// Estatísticas de comunicações com a JIGA07
	statJIGA07_Comunicacao : statistics_int;
	// Variável utilizada para registros
	iJIGA01_LastTempoSemComunicacao : INT := 30000;
	// Variável utilizada para registros
	iJIGA02_LastTempoSemComunicacao : INT := 30000;
	// Variável utilizada para registros
	iJIGA03_LastTempoSemComunicacao : INT := 30000;
	// Variável utilizada para registros
	iJIGA05_LastTempoSemComunicacao : INT := 30000;
	// Variável utilizada para registros
	iJIGA07_LastTempoSemComunicacao : INT := 30000;
	// Variável utilizada para registros
	wJIGA01_Estatistica_QtdComRasc : WORD;
	// Variável utilizada para registros
	wJIGA02_Estatistica_QtdComRasc : WORD;
	// Variável utilizada para registros
	wJIGA03_Estatistica_QtdComRasc : WORD;
	// Variável utilizada para registros
	wJIGA05_Estatistica_QtdComRasc : WORD;
	// Variável utilizada para registros
	wJIGA07_Estatistica_QtdComRasc : WORD;
	// Variável que mostra a quantidade de comunicações que houveram com a JIGA01
	lwJIGA01_Estatistica_QtdCom : LWORD;
	// Variável que mostra a quantidade de comunicações que houveram com a JIGA02
	lwJIGA02_Estatistica_QtdCom : LWORD;
	// Variável que mostra a quantidade de comunicações que houveram com a JIGA03
	lwJIGA03_Estatistica_QtdCom : LWORD;
	// Variável que mostra a quantidade de comunicações que houveram com a JIGA05
	lwJIGA05_Estatistica_QtdCom : LWORD;
	// Variável que mostra a quantidade de comunicações que houveram com a JIGA07
	lwJIGA07_Estatistica_QtdCom : LWORD;
	tTimerRetainCleanStatus : TON;
	// Resultados da comunicação com a JIGA01
	{attribute 'symbol' := 'read'}
	JIGA01 : NVL_Result;
	// Resultados da comunicação com a JIGA02
	{attribute 'symbol' := 'read'}
	JIGA02 : NVL_Result;
	// Resultados da comunicação com a JIGA03
	{attribute 'symbol' := 'read'}
	JIGA03 : NVL_Result;
	// Resultados da comunicação com a JIGA05
	{attribute 'symbol' := 'read'}
	JIGA05 : NVL_Result;
	// Resultados da comunicação com a JIGA07
	{attribute 'symbol' := 'read'}
	JIGA07 : NVL_Result;
	uliPouIniTime : ULINT;
	uliPouEndTime : ULINT;
END_VAR

//*****************************************************************************
// Autor(es): Roberto Martiny
// Descrição:
// POU para consistência da funcionalidade NVL 
//*****************************************************************************

// Registra o tempo do sistema
SysTimeGetUs(uliPouIniTime);


// Contador para informar as outras NVLs que este CP está  funcionando. 
NVL_Sender_BroadCast_for_all.iKeepAlive_JIGA03b:= NVL_Sender_BroadCast_for_all.iKeepAlive_JIGA03b+1;

//*******************************************************************************************************************************************************
// Testa comunicação entre JIGA 03 e JIGA 01
//*******************************************************************************************************************************************************
// Se valor recebido for igual ao enviado...
IF NVL_Sender_JIGA03_Exclusive_to_JIGA01.iJIGA03_TO_JIGA01e= NVL_Receiver_JIGA01_Broadcast.iJIGA01_TO_JIGA03b THEN
	// Incrementa contador para próximo teste
	NVL_Sender_JIGA03_Exclusive_to_JIGA01.iJIGA03_TO_JIGA01e:= NVL_Sender_JIGA03_Exclusive_to_JIGA01.iJIGA03_TO_JIGA01e+1;
	// Se próximo valor do contador for igual ao valor da constante utilizada para informar que houve um CleanTest, pula esse valor 
	IF NVL_Sender_JIGA03_Exclusive_to_JIGA01.iJIGA03_TO_JIGA01e = ProjectConstants.iNVL_CleanTest THEN
		NVL_Sender_JIGA03_Exclusive_to_JIGA01.iJIGA03_TO_JIGA01e:= 0;
	END_IF
	// Sempre que houver sucesso na comunicação zera contador de ciclos
	iJIGA01_CiclosSemComunicao:=0;
ELSE
	// Enquanto o valor do retorno não for o esperado, incrementa contador de ciclos
	iJIGA01_CiclosSemComunicao:= iJIGA01_CiclosSemComunicao+1;
	IF iJIGA01_CiclosSemComunicao*ProjectConstants.iMainTaskInterval > 30000 THEN
		iJIGA01_CiclosSemComunicao:=30000/ProjectConstants.iMainTaskInterval;
	END_IF
END_IF
// Se o tempo for maior que o tempo esperado, liga flag de erro
IF iJIGA01_CiclosSemComunicao*ProjectConstants.iMainTaskInterval > ProjectConstants.iNVL_MaximumInterval THEN
	PersistentVars.bFailNVLCommunicationJIGA01:= TRUE;
END_IF
// Caso receba o valor de constante informando que houve um CleanTest na outra jiga, reincia diagnósticos e estatísticas desta jiga
IF NVL_Receiver_JIGA01_Broadcast.iJIGA01_TO_JIGA03b = ProjectConstants.iNVL_CleanTest THEN
	ctuJIGA01_QtdComunicao.RESET := TRUE;
	ctuJIGA01_QtdComunicao3s.RESET := TRUE;
	ctuJIGA01_QtdComunicao4s.RESET := TRUE;
	ctuJIGA01_QtdComunicao5s.RESET := TRUE;
	statJIGA01_Comunicacao.RESET := TRUE;
	PersistentVars.bFailNVLCommunicationJIGA01:= FALSE;
	iJIGA01_CiclosSemComunicao:= 0;
	iJIGA01_CiclosSemComunicaoMax:= 0;
END_IF
// Faz o retorno do valor recebido da JIGA 01 para a JIGA 03
NVL_Sender_BroadCast_for_all.iJIGA03_TO_JIGA01b:= NVL_Receiver_JIGA01_Exclusive.iJIGA01_TO_JIGA03e;

//*******************************************************************************************************************************************************

//*******************************************************************************************************************************************************
// Testa comunicação entre JIGA 03 e JIGA 02
//*******************************************************************************************************************************************************
// Se valor recebido for igual ao enviado...
IF NVL_Sender_JIGA03_Exclusive_to_JIGA02.iJIGA03_TO_JIGA02e= NVL_Receiver_JIGA02_Broadcast.iJIGA02_TO_JIGA03b THEN
	// Incrementa contador para próximo teste
	NVL_Sender_JIGA03_Exclusive_to_JIGA02.iJIGA03_TO_JIGA02e:= NVL_Sender_JIGA03_Exclusive_to_JIGA02.iJIGA03_TO_JIGA02e+1;
	// Se próximo valor do contador for igual ao valor da constante utilizada para informar que houve um CleanTest, pula esse valor 
	IF NVL_Sender_JIGA03_Exclusive_to_JIGA02.iJIGA03_TO_JIGA02e = ProjectConstants.iNVL_CleanTest THEN
		NVL_Sender_JIGA03_Exclusive_to_JIGA02.iJIGA03_TO_JIGA02e:= 0;
	END_IF
	// Sempre que houver sucesso na comunicação zera contador de ciclos
	iJIGA02_CiclosSemComunicao:=0;
ELSE
	// Enquanto o valor do retorno não for o esperado, incrementa contador de ciclos
	iJIGA02_CiclosSemComunicao:= iJIGA02_CiclosSemComunicao+1;
	IF iJIGA02_CiclosSemComunicao*ProjectConstants.iMainTaskInterval > 30000 THEN
		iJIGA02_CiclosSemComunicao:=30000/ProjectConstants.iMainTaskInterval;
	END_IF
END_IF
// Se o tempo for maior que o tempo esperado, liga flag de erro
IF iJIGA02_CiclosSemComunicao*ProjectConstants.iMainTaskInterval > ProjectConstants.iNVL_MaximumInterval THEN
	PersistentVars.bFailNVLCommunicationJIGA02:= TRUE;
END_IF
// Caso receba o valor de constante informando que houve um CleanTest na outra jiga, reincia diagnósticos e estatísticas desta jiga
IF NVL_Receiver_JIGA02_Broadcast.iJIGA02_TO_JIGA03b = ProjectConstants.iNVL_CleanTest THEN
	ctuJIGA02_QtdComunicao.RESET := TRUE;
	ctuJIGA02_QtdComunicao3s.RESET := TRUE;
	ctuJIGA02_QtdComunicao4s.RESET := TRUE;
	ctuJIGA02_QtdComunicao5s.RESET := TRUE;
	statJIGA02_Comunicacao.RESET := TRUE;
	PersistentVars.bFailNVLCommunicationJIGA02:= FALSE;
	iJIGA02_CiclosSemComunicao:= 0;
	iJIGA02_CiclosSemComunicaoMax:= 0;
END_IF
// Faz o retorno do valor recebido da JIGA 02 para a JIGA 03
NVL_Sender_BroadCast_for_all.iJIGA03_TO_JIGA02b:= NVL_Receiver_JIGA02_Exclusive.iJIGA02_TO_JIGA03e;

//*******************************************************************************************************************************************************

//*******************************************************************************************************************************************************
// Testa comunicação entre JIGA03 e JIGA05
//*******************************************************************************************************************************************************
// Se valor recebido for igual ao enviado...
IF NVL_Sender_JIGA03_Exclusive_to_JIGA05.iJIGA03_TO_JIGA05e= NVL_Receiver_JIGA05_Broadcast.iJIGA05_TO_JIGA03b THEN
	// Incrementa contador para próximo teste
	NVL_Sender_JIGA03_Exclusive_to_JIGA05.iJIGA03_TO_JIGA05e:= NVL_Sender_JIGA03_Exclusive_to_JIGA05.iJIGA03_TO_JIGA05e+1;
	// Se próximo valor do contador for igual ao valor da constante utilizada para informar que houve um CleanTest, pula esse valor 
	IF NVL_Sender_JIGA03_Exclusive_to_JIGA05.iJIGA03_TO_JIGA05e = ProjectConstants.iNVL_CleanTest THEN
		NVL_Sender_JIGA03_Exclusive_to_JIGA05.iJIGA03_TO_JIGA05e:= 0;
	END_IF
	// Sempre que houver sucesso na comunicação zera contador de ciclos
	iJIGA05_CiclosSemComunicao:=0;
ELSE
	// Enquanto o valor do retorno não for o esperado, incrementa contador de ciclos
	iJIGA05_CiclosSemComunicao:= iJIGA05_CiclosSemComunicao+1;
	IF iJIGA05_CiclosSemComunicao*ProjectConstants.iMainTaskInterval > 30000 THEN
		iJIGA05_CiclosSemComunicao:=30000/ProjectConstants.iMainTaskInterval;
	END_IF
END_IF
// Se o tempo for maior que o tempo esperado, liga flag de erro
IF iJIGA05_CiclosSemComunicao*ProjectConstants.iMainTaskInterval > ProjectConstants.iNVL_MaximumInterval THEN
	PersistentVars.bFailNVLCommunicationJIGA05:= TRUE;
END_IF
// Caso receba o valor de constante informando que houve um CleanTest na outra jiga, reincia diagnósticos e estatísticas desta jiga
IF NVL_Receiver_JIGA05_Broadcast.iJIGA05_TO_JIGA03b = ProjectConstants.iNVL_CleanTest THEN
	ctuJIGA05_QtdComunicao.RESET := TRUE;
	ctuJIGA05_QtdComunicao3s.RESET := TRUE;
	ctuJIGA05_QtdComunicao4s.RESET := TRUE;
	ctuJIGA05_QtdComunicao5s.RESET := TRUE;
	statJIGA05_Comunicacao.RESET := TRUE;
	PersistentVars.bFailNVLCommunicationJIGA05:= FALSE;
	iJIGA05_CiclosSemComunicao:= 0;
	iJIGA05_CiclosSemComunicaoMax:= 0;
END_IF
// Faz o retorno do valor recebido da JIGA05 para a JIGA03
NVL_Sender_BroadCast_for_all.iJIGA03_TO_JIGA05b:= NVL_Receiver_JIGA05_Exclusive.iJIGA05_TO_JIGA03e;

//*******************************************************************************************************************************************************

//*******************************************************************************************************************************************************
// Testa comunicação entre JIGA03 e JIGA07
//*******************************************************************************************************************************************************
// Se valor recebido for igual ao enviado...
IF NVL_Sender_JIGA03_Exclusive_to_JIGA07.iJIGA03_TO_JIGA07e= NVL_Receiver_JIGA07_Broadcast.iJIGA07_TO_JIGA03b THEN
	// Incrementa contador para próximo teste
	NVL_Sender_JIGA03_Exclusive_to_JIGA07.iJIGA03_TO_JIGA07e:= NVL_Sender_JIGA03_Exclusive_to_JIGA07.iJIGA03_TO_JIGA07e+1;
	// Se próximo valor do contador for igual ao valor da constante utilizada para informar que houve um CleanTest, pula esse valor 
	IF NVL_Sender_JIGA03_Exclusive_to_JIGA07.iJIGA03_TO_JIGA07e = ProjectConstants.iNVL_CleanTest THEN
		NVL_Sender_JIGA03_Exclusive_to_JIGA07.iJIGA03_TO_JIGA07e:= 0;
	END_IF
	// Sempre que houver sucesso na comunicação zera contador de ciclos
	iJIGA07_CiclosSemComunicao:=0;
ELSE
	// Enquanto o valor do retorno não for o esperado, incrementa contador de ciclos
	iJIGA07_CiclosSemComunicao:= iJIGA07_CiclosSemComunicao+1;
	IF iJIGA07_CiclosSemComunicao*ProjectConstants.iMainTaskInterval > 30000 THEN
		iJIGA07_CiclosSemComunicao:=30000/ProjectConstants.iMainTaskInterval;
	END_IF
END_IF
// Se o tempo for maior que o tempo esperado, liga flag de erro
IF iJIGA07_CiclosSemComunicao*ProjectConstants.iMainTaskInterval > ProjectConstants.iNVL_MaximumInterval THEN
	PersistentVars.bFailNVLCommunicationJIGA07:= TRUE;
END_IF
// Caso receba o valor de constante informando que houve um CleanTest na outra jiga, reincia diagnósticos e estatísticas desta jiga
IF NVL_Receiver_JIGA07_Broadcast.iJIGA07_TO_JIGA03b = ProjectConstants.iNVL_CleanTest THEN
	ctuJIGA07_QtdComunicao.RESET := TRUE;
	ctuJIGA07_QtdComunicao3s.RESET := TRUE;
	ctuJIGA07_QtdComunicao4s.RESET := TRUE;
	ctuJIGA07_QtdComunicao5s.RESET := TRUE;
	statJIGA07_Comunicacao.RESET := TRUE;
	PersistentVars.bFailNVLCommunicationJIGA07:= FALSE;
	iJIGA07_CiclosSemComunicao:= 0;
	iJIGA07_CiclosSemComunicaoMax:= 0;
END_IF
// Faz o retorno do valor recebido da JIGA07 para a JIGA03
NVL_Sender_BroadCast_for_all.iJIGA03_TO_JIGA07b:= NVL_Receiver_JIGA07_Exclusive.iJIGA07_TO_JIGA03e;

//*******************************************************************************************************************************************************


//*******************************************************************************************************************************************************
// Estatísticas da Comunicação
//*******************************************************************************************************************************************************

// JIGA01
// Contador de Quantidades de Comunicações realizadas
IF iJIGA01_CiclosSemComunicao = 0 THEN
	ctuJIGA01_QtdComunicao.CU:= TRUE;
	statJIGA01_Comunicacao.IN:=iJIGA01_LastTempoSemComunicacao;
	statJIGA01_Comunicacao();
	statJIGA01_Comunicacao.RESET := FALSE;
ELSE
	ctuJIGA01_QtdComunicao.CU:= FALSE;
	// Cópia do ultimo tempo para comunicação
	iJIGA01_LastTempoSemComunicacao:= iJIGA01_CiclosSemComunicao*ProjectConstants.iMainTaskInterval;
END_IF
ctuJIGA01_QtdComunicao();
ctuJIGA01_QtdComunicao.RESET := FALSE;
IF ctuJIGA01_QtdComunicao.CV = 60000 THEN
	wJIGA01_Estatistica_QtdComRasc:=wJIGA01_Estatistica_QtdComRasc+1;
	ctuJIGA01_QtdComunicao.RESET := TRUE;
END_IF
lwJIGA01_Estatistica_QtdCom:= wJIGA01_Estatistica_QtdComRasc*60000+ ctuJIGA01_QtdComunicao.CV;

// Contador de Quantidades de Comunicações acimade 3 segundos
IF iJIGA01_CiclosSemComunicao > 3000/ProjectConstants.iMainTaskInterval THEN
	ctuJIGA01_QtdComunicao3s.CU:= TRUE;
ELSE
	ctuJIGA01_QtdComunicao3s.CU:= FALSE;
END_IF
ctuJIGA01_QtdComunicao3s();
ctuJIGA01_QtdComunicao3s.RESET := FALSE;

// Contador de Quantidades de Comunicações acimade 4 segundos
IF iJIGA01_CiclosSemComunicao > 4000/ProjectConstants.iMainTaskInterval THEN
	ctuJIGA01_QtdComunicao4s.CU:= TRUE;
ELSE
	ctuJIGA01_QtdComunicao4s.CU:= FALSE;
END_IF
ctuJIGA01_QtdComunicao4s();
ctuJIGA01_QtdComunicao4s.RESET:=FALSE;

// Contador de Quantidades de Comunicações acimade 5 segundos
IF iJIGA01_CiclosSemComunicao > 5000/ProjectConstants.iMainTaskInterval THEN
	ctuJIGA01_QtdComunicao5s.CU:= TRUE;
ELSE
	ctuJIGA01_QtdComunicao5s.CU:= FALSE;
END_IF
ctuJIGA01_QtdComunicao5s();
ctuJIGA01_QtdComunicao5s.RESET := FALSE;


JIGA01.iTempoMinimo:= statJIGA01_Comunicacao.MN;
JIGA01.iTempoMedio:= statJIGA01_Comunicacao.AVG;
JIGA01.iTempoMaximo:= statJIGA01_Comunicacao.MX;
JIGA01.lwQtdTotalComunicacoes:= lwJIGA01_Estatistica_QtdCom;
JIGA01.wQtdComMaior3segundos:= ctuJIGA01_QtdComunicao3s.CV;
JIGA01.wQtdComMaior4segundos:= ctuJIGA01_QtdComunicao4s.CV;
JIGA01.wQtdComMaior5segundos:= ctuJIGA01_QtdComunicao5s.CV;

// JIGA02
// Contador de Quantidades de Comunicações realizadas
IF iJIGA02_CiclosSemComunicao = 0 THEN
	ctuJIGA02_QtdComunicao.CU:= TRUE;
	statJIGA02_Comunicacao.IN:=iJIGA02_LastTempoSemComunicacao;
	statJIGA02_Comunicacao();
	statJIGA02_Comunicacao.RESET := FALSE;
ELSE
	ctuJIGA02_QtdComunicao.CU:= FALSE;
	// Cópia do ultimo tempo para comunicação
	iJIGA02_LastTempoSemComunicacao:= iJIGA02_CiclosSemComunicao*ProjectConstants.iMainTaskInterval;
END_IF
ctuJIGA02_QtdComunicao();
ctuJIGA02_QtdComunicao.RESET := FALSE;
IF ctuJIGA02_QtdComunicao.CV = 60000 THEN
	wJIGA02_Estatistica_QtdComRasc:=wJIGA02_Estatistica_QtdComRasc+1;
	ctuJIGA02_QtdComunicao.RESET := TRUE;
END_IF
lwJIGA02_Estatistica_QtdCom:= wJIGA02_Estatistica_QtdComRasc*60000+ ctuJIGA02_QtdComunicao.CV;

// Contador de Quantidades de Comunicações acimade 3 segundos
IF iJIGA02_CiclosSemComunicao > 3000/ProjectConstants.iMainTaskInterval THEN
	ctuJIGA02_QtdComunicao3s.CU:= TRUE;
ELSE
	ctuJIGA02_QtdComunicao3s.CU:= FALSE;
END_IF
ctuJIGA02_QtdComunicao3s();
ctuJIGA02_QtdComunicao3s.RESET := FALSE;

// Contador de Quantidades de Comunicações acimade 4 segundos
IF iJIGA02_CiclosSemComunicao > 4000/ProjectConstants.iMainTaskInterval THEN
	ctuJIGA02_QtdComunicao4s.CU:= TRUE;
ELSE
	ctuJIGA02_QtdComunicao4s.CU:= FALSE;
END_IF
ctuJIGA02_QtdComunicao4s();
ctuJIGA02_QtdComunicao4s.RESET:=FALSE;

// Contador de Quantidades de Comunicações acimade 5 segundos
IF iJIGA02_CiclosSemComunicao > 5000/ProjectConstants.iMainTaskInterval THEN
	ctuJIGA02_QtdComunicao5s.CU:= TRUE;
ELSE
	ctuJIGA02_QtdComunicao5s.CU:= FALSE;
END_IF
ctuJIGA02_QtdComunicao5s();
ctuJIGA02_QtdComunicao5s.RESET := FALSE;

JIGA02.iTempoMinimo:= statJIGA02_Comunicacao.MN;
JIGA02.iTempoMedio:= statJIGA02_Comunicacao.AVG;
JIGA02.iTempoMaximo:= statJIGA02_Comunicacao.MX;
JIGA02.lwQtdTotalComunicacoes:= lwJIGA02_Estatistica_QtdCom;
JIGA02.wQtdComMaior3segundos:= ctuJIGA02_QtdComunicao3s.CV;
JIGA02.wQtdComMaior4segundos:= ctuJIGA02_QtdComunicao4s.CV;
JIGA02.wQtdComMaior5segundos:= ctuJIGA02_QtdComunicao5s.CV;

// JIGA03
// Contador de Quantidades de Comunicações realizadas
IF iJIGA03_CiclosSemComunicao = 0 THEN
	ctuJIGA03_QtdComunicao.CU:= TRUE;
	statJIGA03_Comunicacao.IN:=iJIGA03_LastTempoSemComunicacao;
	statJIGA03_Comunicacao();
	statJIGA03_Comunicacao.RESET := FALSE;
ELSE
	ctuJIGA03_QtdComunicao.CU:= FALSE;
	// Cópia do ultimo tempo para comunicação
	iJIGA03_LastTempoSemComunicacao:= iJIGA03_CiclosSemComunicao*ProjectConstants.iMainTaskInterval;
END_IF
ctuJIGA03_QtdComunicao();
ctuJIGA03_QtdComunicao.RESET := FALSE;
IF ctuJIGA03_QtdComunicao.CV = 60000 THEN
	wJIGA03_Estatistica_QtdComRasc:=wJIGA03_Estatistica_QtdComRasc+1;
	ctuJIGA03_QtdComunicao.RESET := TRUE;
END_IF
lwJIGA03_Estatistica_QtdCom:= wJIGA03_Estatistica_QtdComRasc*60000+ ctuJIGA03_QtdComunicao.CV;

// Contador de Quantidades de Comunicações acimade 3 segundos
IF iJIGA03_CiclosSemComunicao > 3000/ProjectConstants.iMainTaskInterval THEN
	ctuJIGA03_QtdComunicao3s.CU:= TRUE;
ELSE
	ctuJIGA03_QtdComunicao3s.CU:= FALSE;
END_IF
ctuJIGA03_QtdComunicao3s();
ctuJIGA03_QtdComunicao3s.RESET := FALSE;

// Contador de Quantidades de Comunicações acimade 4 segundos
IF iJIGA03_CiclosSemComunicao > 4000/ProjectConstants.iMainTaskInterval THEN
	ctuJIGA03_QtdComunicao4s.CU:= TRUE;
ELSE
	ctuJIGA03_QtdComunicao4s.CU:= FALSE;
END_IF
ctuJIGA03_QtdComunicao4s();
ctuJIGA03_QtdComunicao4s.RESET:=FALSE;

// Contador de Quantidades de Comunicações acimade 5 segundos
IF iJIGA03_CiclosSemComunicao > 5000/ProjectConstants.iMainTaskInterval THEN
	ctuJIGA03_QtdComunicao5s.CU:= TRUE;
ELSE
	ctuJIGA03_QtdComunicao5s.CU:= FALSE;
END_IF
ctuJIGA03_QtdComunicao5s();
ctuJIGA03_QtdComunicao5s.RESET := FALSE;

JIGA03.iTempoMinimo:= statJIGA03_Comunicacao.MN;
JIGA03.iTempoMedio:= statJIGA03_Comunicacao.AVG;
JIGA03.iTempoMaximo:= statJIGA03_Comunicacao.MX;
JIGA03.lwQtdTotalComunicacoes:= lwJIGA03_Estatistica_QtdCom;
JIGA03.wQtdComMaior3segundos:= ctuJIGA03_QtdComunicao3s.CV;
JIGA03.wQtdComMaior4segundos:= ctuJIGA03_QtdComunicao4s.CV;
JIGA03.wQtdComMaior5segundos:= ctuJIGA03_QtdComunicao5s.CV;

// JIGA05
// Contador de Quantidades de Comunicações realizadas
IF iJIGA05_CiclosSemComunicao = 0 THEN
	ctuJIGA05_QtdComunicao.CU:= TRUE;
	statJIGA05_Comunicacao.IN:=iJIGA05_LastTempoSemComunicacao;
	statJIGA05_Comunicacao();
	statJIGA05_Comunicacao.RESET := FALSE;
ELSE
	ctuJIGA05_QtdComunicao.CU:= FALSE;
	// Cópia do ultimo tempo para comunicação
	iJIGA05_LastTempoSemComunicacao:= iJIGA05_CiclosSemComunicao*ProjectConstants.iMainTaskInterval;
END_IF
ctuJIGA05_QtdComunicao();
ctuJIGA05_QtdComunicao.RESET := FALSE;
IF ctuJIGA05_QtdComunicao.CV = 60000 THEN
	wJIGA05_Estatistica_QtdComRasc:=wJIGA05_Estatistica_QtdComRasc+1;
	ctuJIGA05_QtdComunicao.RESET := TRUE;
END_IF
lwJIGA05_Estatistica_QtdCom:= wJIGA05_Estatistica_QtdComRasc*60000+ ctuJIGA05_QtdComunicao.CV;

// Contador de Quantidades de Comunicações acimade 3 segundos
IF iJIGA05_CiclosSemComunicao > 3000/ProjectConstants.iMainTaskInterval THEN
	ctuJIGA05_QtdComunicao3s.CU:= TRUE;
ELSE
	ctuJIGA05_QtdComunicao3s.CU:= FALSE;
END_IF
ctuJIGA05_QtdComunicao3s();
ctuJIGA05_QtdComunicao3s.RESET := FALSE;

// Contador de Quantidades de Comunicações acimade 4 segundos
IF iJIGA05_CiclosSemComunicao > 4000/ProjectConstants.iMainTaskInterval THEN
	ctuJIGA05_QtdComunicao4s.CU:= TRUE;
ELSE
	ctuJIGA05_QtdComunicao4s.CU:= FALSE;
END_IF
ctuJIGA05_QtdComunicao4s();
ctuJIGA05_QtdComunicao4s.RESET:=FALSE;

// Contador de Quantidades de Comunicações acimade 5 segundos
IF iJIGA05_CiclosSemComunicao > 5000/ProjectConstants.iMainTaskInterval THEN
	ctuJIGA05_QtdComunicao5s.CU:= TRUE;
ELSE
	ctuJIGA05_QtdComunicao5s.CU:= FALSE;
END_IF
ctuJIGA05_QtdComunicao5s();
ctuJIGA05_QtdComunicao5s.RESET := FALSE;

JIGA05.iTempoMinimo:= statJIGA05_Comunicacao.MN;
JIGA05.iTempoMedio:= statJIGA05_Comunicacao.AVG;
JIGA05.iTempoMaximo:= statJIGA05_Comunicacao.MX;
JIGA05.lwQtdTotalComunicacoes:= lwJIGA05_Estatistica_QtdCom;
JIGA05.wQtdComMaior3segundos:= ctuJIGA05_QtdComunicao3s.CV;
JIGA05.wQtdComMaior4segundos:= ctuJIGA05_QtdComunicao4s.CV;
JIGA05.wQtdComMaior5segundos:= ctuJIGA05_QtdComunicao5s.CV;

// JIGA07
// Contador de Quantidades de Comunicações realizadas
IF iJIGA07_CiclosSemComunicao = 0 THEN
	ctuJIGA07_QtdComunicao.CU:= TRUE;
	statJIGA07_Comunicacao.IN:=iJIGA07_LastTempoSemComunicacao;
	statJIGA07_Comunicacao();
	statJIGA07_Comunicacao.RESET := FALSE;
ELSE
	ctuJIGA07_QtdComunicao.CU:= FALSE;
	// Cópia do ultimo tempo para comunicação
	iJIGA07_LastTempoSemComunicacao:= iJIGA07_CiclosSemComunicao*ProjectConstants.iMainTaskInterval;
END_IF
ctuJIGA07_QtdComunicao();
ctuJIGA07_QtdComunicao.RESET := FALSE;
IF ctuJIGA07_QtdComunicao.CV = 60000 THEN
	wJIGA07_Estatistica_QtdComRasc:=wJIGA07_Estatistica_QtdComRasc+1;
	ctuJIGA07_QtdComunicao.RESET := TRUE;
END_IF
lwJIGA07_Estatistica_QtdCom:= wJIGA07_Estatistica_QtdComRasc*60000+ ctuJIGA07_QtdComunicao.CV;

// Contador de Quantidades de Comunicações acimade 3 segundos
IF iJIGA07_CiclosSemComunicao > 3000/ProjectConstants.iMainTaskInterval THEN
	ctuJIGA07_QtdComunicao3s.CU:= TRUE;
ELSE
	ctuJIGA07_QtdComunicao3s.CU:= FALSE;
END_IF
ctuJIGA07_QtdComunicao3s();
ctuJIGA07_QtdComunicao3s.RESET := FALSE;

// Contador de Quantidades de Comunicações acimade 4 segundos
IF iJIGA07_CiclosSemComunicao > 4000/ProjectConstants.iMainTaskInterval THEN
	ctuJIGA07_QtdComunicao4s.CU:= TRUE;
ELSE
	ctuJIGA07_QtdComunicao4s.CU:= FALSE;
END_IF
ctuJIGA07_QtdComunicao4s();
ctuJIGA07_QtdComunicao4s.RESET:=FALSE;

// Contador de Quantidades de Comunicações acimade 5 segundos
IF iJIGA07_CiclosSemComunicao > 5000/ProjectConstants.iMainTaskInterval THEN
	ctuJIGA07_QtdComunicao5s.CU:= TRUE;
ELSE
	ctuJIGA07_QtdComunicao5s.CU:= FALSE;
END_IF
ctuJIGA07_QtdComunicao5s();
ctuJIGA07_QtdComunicao5s.RESET := FALSE;

JIGA07.iTempoMinimo:= statJIGA07_Comunicacao.MN;
JIGA07.iTempoMedio:= statJIGA07_Comunicacao.AVG;
JIGA07.iTempoMaximo:= statJIGA07_Comunicacao.MX;
JIGA07.lwQtdTotalComunicacoes:= lwJIGA07_Estatistica_QtdCom;
JIGA07.wQtdComMaior3segundos:= ctuJIGA07_QtdComunicao3s.CV;
JIGA07.wQtdComMaior4segundos:= ctuJIGA07_QtdComunicao4s.CV;
JIGA07.wQtdComMaior5segundos:= ctuJIGA07_QtdComunicao5s.CV;

//*******************************************************************************************************************************************************

//*******************************************************************************************************************************************************
// Se for gerado um comando de CleanStats nesta jiga, envia constante que informa isso para as outras jigas reiniciarem suas estatítitcas e 
// diagnósticos com esse jiga
IF Symbolics.bEnableCleanStats_CheckNVL THEN
	
	ctuJIGA01_QtdComunicao.RESET := TRUE;
	ctuJIGA02_QtdComunicao.RESET := TRUE;
	ctuJIGA03_QtdComunicao.RESET := TRUE;
	ctuJIGA05_QtdComunicao.RESET := TRUE;
	ctuJIGA07_QtdComunicao.RESET := TRUE;
	ctuJIGA01_QtdComunicao3s.RESET := TRUE;
	ctuJIGA02_QtdComunicao3s.RESET := TRUE;
	ctuJIGA03_QtdComunicao3s.RESET := TRUE;
	ctuJIGA05_QtdComunicao3s.RESET := TRUE;
	ctuJIGA07_QtdComunicao3s.RESET := TRUE;
	ctuJIGA01_QtdComunicao4s.RESET := TRUE;
	ctuJIGA02_QtdComunicao4s.RESET := TRUE;
	ctuJIGA03_QtdComunicao4s.RESET := TRUE;
	ctuJIGA05_QtdComunicao4s.RESET := TRUE;
	ctuJIGA07_QtdComunicao4s.RESET := TRUE;
	ctuJIGA01_QtdComunicao5s.RESET := TRUE;
	ctuJIGA02_QtdComunicao5s.RESET := TRUE;
	ctuJIGA03_QtdComunicao5s.RESET := TRUE;
	ctuJIGA05_QtdComunicao5s.RESET := TRUE;
	ctuJIGA07_QtdComunicao5s.RESET := TRUE;
	statJIGA01_Comunicacao.RESET := TRUE;
	statJIGA02_Comunicacao.RESET := TRUE;
	statJIGA03_Comunicacao.RESET := TRUE;
	statJIGA05_Comunicacao.RESET := TRUE;
	statJIGA07_Comunicacao.RESET := TRUE;
		
	PersistentVars.bFailNVLCommunicationJIGA01:= FALSE;
	PersistentVars.bFailNVLCommunicationJIGA02:= FALSE;
	PersistentVars.bFailNVLCommunicationJIGA05:= FALSE;
	PersistentVars.bFailNVLCommunicationJIGA07:= FALSE;

	
	iJIGA01_CiclosSemComunicao:= 0;
	iJIGA02_CiclosSemComunicao:= 0;
	iJIGA03_CiclosSemComunicao:= 0;
	iJIGA05_CiclosSemComunicao:= 0;
	iJIGA07_CiclosSemComunicao:= 0;
	
	iJIGA01_CiclosSemComunicaoMax:= 0;
	iJIGA02_CiclosSemComunicaoMax:= 0;
	iJIGA03_CiclosSemComunicaoMax:= 0;
	iJIGA05_CiclosSemComunicaoMax:= 0;
	iJIGA07_CiclosSemComunicaoMax:= 0;

	// Código para comando de CleanStats
	NVL_Sender_BroadCast_for_all.iJIGA03_TO_JIGA01b := -1;
	NVL_Sender_BroadCast_for_all.iJIGA03_TO_JIGA02b := -1;
	NVL_Sender_BroadCast_for_all.iJIGA03_TO_JIGA05b := -1;
	NVL_Sender_BroadCast_for_all.iJIGA03_TO_JIGA07b := -1;
	
	// Mantém essa escrita pelo tempo comfigurado abaixo (tempo do poolingo configurado para o NVL)
	tTimerRetainCleanStatus.PT:=T#2S;
	tTimerRetainCleanStatus();
	tTimerRetainCleanStatus.IN:=TRUE;
	IF tTimerRetainCleanStatus.Q THEN
		Symbolics.bEnableCleanStats_CheckNVL:= FALSE;	
		tTimerRetainCleanStatus.IN:= FALSE;
	END_IF
END_IF
//*******************************************************************************************************************************************************

// Registra o tempo do sistema
SysTimeGetUs(uliPouEndTime);
// Calcula duração mínima/máxima desta POU
MinMaxTimes.uliPouMinTime_CheckNVL:= MIN(MinMaxTimes.uliPouMinTime_CheckNVL, uliPouEndTime - uliPouIniTime);
MinMaxTimes.uliPouMaxTime_CheckNVL:= MAX(MinMaxTimes.uliPouMaxTime_CheckNVL, uliPouEndTime - uliPouIniTime);

END_PROGRAM

// Device/Application/UserPOUs/Redundant/IncrRedData
PROGRAM IncrRedData
VAR
	dwIndex : DWORD;
	ptIW : POINTER TO INT;
	// Depuração dos tempos dos laços
	maxdiff : ARRAY [0..6] OF systime;
	// Depuração dos tempos dos laços
	tempo : ARRAY [0..6] OF systime;
	// Depuração dos tempos dos laços
	diff : ARRAY [0..6] OF systime;
	uliPouIniTime : ULINT;
	uliPouEndTime : ULINT;
END_VAR

// Escreve valores em todas as variáveis de dados redundantes

// Registra o tempo do sistema
SysTimeGetUs(uliPouIniTime);

tempo[0]:= SysTimeGetMs();

// Incrementa o valor das variáveis redundantes
IF Symbolics.iValueRed >= ProjectConstants.iValueRedLimit THEN
	Symbolics.iValueRed:= 1;
ELSE
	Symbolics.iValueRed:= Symbolics.iValueRed + 1;
END_IF

// Incrementa o array simbólico
FOR dwIndex:= 1 TO (SIZEOF(Symbolics.aiRedundantArrayS)/SIZEOF(Symbolics.aiRedundantArrayS[1])) DO
	Symbolics.aiRedundantArrayS[dwIndex]:= Symbolics.iValueRed;
END_FOR
FOR dwIndex:= 1 TO (SIZEOF(Symbolics.aiRedundantArrayS1)/SIZEOF(Symbolics.aiRedundantArrayS1[1])) DO
	Symbolics.aiRedundantArrayS1[dwIndex]:= Symbolics.iValueRed;
END_FOR
FOR dwIndex:= 1 TO (SIZEOF(Symbolics.aiRedundantArrayS2)/SIZEOF(Symbolics.aiRedundantArrayS2[1])) DO
	Symbolics.aiRedundantArrayS2[dwIndex]:= Symbolics.iValueRed;
END_FOR
FOR dwIndex:= 1 TO (SIZEOF(Symbolics.aiRedundantArrayS3)/SIZEOF(Symbolics.aiRedundantArrayS3[1])) DO
	Symbolics.aiRedundantArrayS3[dwIndex]:= Symbolics.iValueRed;
END_FOR
FOR dwIndex:= 1 TO (SIZEOF(Symbolics.aiRedundantArrayS4)/SIZEOF(Symbolics.aiRedundantArrayS4[1])) DO
	Symbolics.aiRedundantArrayS4[dwIndex]:= Symbolics.iValueRed;
END_FOR
tempo[1]:= SysTimeGetMs();

// Incrementa o array AT %Q
FOR dwIndex:= 1 TO (SIZEOF(ATs.aiRedundantArrayQ)/SIZEOF(ATs.aiRedundantArrayQ[1])) DO
	ATs.aiRedundantArrayQ[dwIndex]:= Symbolics.iValueRed;
END_FOR
FOR dwIndex:= 1 TO (SIZEOF(ATs.aiRedundantArrayQ1)/SIZEOF(ATs.aiRedundantArrayQ1[1])) DO
	ATs.aiRedundantArrayQ1[dwIndex]:= Symbolics.iValueRed;
END_FOR

tempo[2]:= SysTimeGetMs();

// Incrementa o array AT %M
FOR dwIndex:= 1 TO (SIZEOF(ATs.aiRedundantArrayM)/SIZEOF(ATs.aiRedundantArrayM[1])) DO
	ATs.aiRedundantArrayM[dwIndex]:= Symbolics.iValueRed;
END_FOR
FOR dwIndex:= 1 TO (SIZEOF(ATs.aiRedundantArrayM1)/SIZEOF(ATs.aiRedundantArrayM1[1])) DO
	ATs.aiRedundantArrayM1[dwIndex]:= Symbolics.iValueRed;
END_FOR


tempo[3]:= SysTimeGetMs();

// Incrementa o array AT %I
FOR ptIW:= ADR(%IW16384) TO (ADR(%IW16384) + SIZEOF(ATs.aiRedundantArrayI)) BY SIZEOF(ATs.aiRedundantArrayI[1]) DO
	ptIW^:= Symbolics.iValueRed;
END_FOR
FOR ptIW:= ADR(%IW28612) TO (ADR(%IW28612) + SIZEOF(ATs.aiRedundantArrayI1)) BY SIZEOF(ATs.aiRedundantArrayI1[1]) DO
	ptIW^:= Symbolics.iValueRed;
END_FOR

tempo[4]:= SysTimeGetMs();

// Envia os resultados para a GVL
	PersistentVars.iSyncFailCntSymb	:=	NonRedPointer.piSSyncFailLoc^	+	NonRedPointer.piSSyncFailRem^;
	PersistentVars.iSyncFailCntQ	:= NonRedPointer.piQSyncFailLoc^	+	NonRedPointer.piQSyncFailRem^;
	PersistentVars.iSyncFailCntM	:= NonRedPointer.piMSyncFailLoc^	+	NonRedPointer.piMSyncFailRem^;
	PersistentVars.iSyncFailCntI	:= NonRedPointer.piISyncFailLoc^	+	NonRedPointer.piISyncFailRem^;


// Cálculo do tempo para execução dos laços
tempo[5] := SysTimeGetMs();
diff[0] := tempo[1] - tempo[0];
diff[1] := tempo[2] - tempo[1];
diff[2] := tempo[3] - tempo[2];
diff[3] := tempo[4] - tempo[3];
diff[4] := tempo[5] - tempo[4];
						
maxdiff[0] := MAX( maxdiff[0], diff[0]);
maxdiff[1] := MAX( maxdiff[1], diff[1]);
maxdiff[2] := MAX( maxdiff[2], diff[2]);
maxdiff[3] := MAX( maxdiff[3], diff[3]);
maxdiff[4] := MAX( maxdiff[4], diff[4]);


// Registra o tempo do sistema
SysTimeGetUs(uliPouEndTime);
// Calcula duração mínima/máxima desta POU
MinMaxTimes.uliPouMinTime_IncrRedData:= MIN(MinMaxTimes.uliPouMinTime_IncrRedData, uliPouEndTime - uliPouIniTime);
MinMaxTimes.uliPouMaxTime_IncrRedData:= MAX(MinMaxTimes.uliPouMaxTime_IncrRedData, uliPouEndTime - uliPouIniTime);

END_PROGRAM

// Device/Application/UserPOUs/Redundant/PidGenerator
PROGRAM PidGenerator
VAR
	state : INT;
	step : REAL := 12;
	uliPouIniTime : ULINT;
	uliPouEndTime : ULINT;
END_VAR

// Gera sinal triangular para estimular o PID Control

// Registra o tempo do sistema
SysTimeGetUs(uliPouIniTime);

// Gera sinal triangular para estimular o PID Control
IF state = 0 THEN
	PIDs.rPID_PV:= PIDs.rPID_PV+step;
	IF PIDs.rPID_PV >20000 THEN
		state := 1;
	END_IF
END_IF

IF state = 1 THEN
	PIDs.rPID_PV:= PIDs.rPID_PV-step;
	IF PIDs.rPID_PV <10000 THEN
		state := 0;
	END_IF
END_IF

// Registra o tempo do sistema
SysTimeGetUs(uliPouEndTime);
// Calcula duração mínima/máxima desta POU
MinMaxTimes.uliPouMinTime_PidGenerator:= MIN(MinMaxTimes.uliPouMinTime_PidGenerator, uliPouEndTime - uliPouIniTime);
MinMaxTimes.uliPouMaxTime_PidGenerator:= MAX(MinMaxTimes.uliPouMaxTime_PidGenerator, uliPouEndTime - uliPouIniTime);

END_PROGRAM

// Device/Application/PIDControl
{attribute 'subsequent'} 
PROGRAM PIDControl
VAR
	MeasureST : BOOL := FALSE;
	NotEqualize : BOOL;

	PV : REAL;
	MV : REAL;

	Controller : NextoPID.PID;
	EffST, Eff3ST, MaxEffST, MinEffST: REAL;
	ErrorCodePID : UINT;
	IntegralAction : REAL;


END_VAR

IF NOT NotEqualize THEN
	IF NOT Manual[1] THEN
		// Automatic mode
		ManualMV[1] := PIDs.rPID_MV;
	END_IF
END_IF

PV := PIDs.rPID_PV;
SP[1] := PIDs.rPID_SP;

Controller(
	SP := PIDs.rPID_SP,
	PV := PIDs.rPID_PV,
	Gp := Gp[1],
	Td := Td[1],
	Ti := Ti[1],
	BIAS := BIAS[1],
	ManualMV := ManualMV[1],
	MaxMV := MaxMV[1],
	MinMV := MinMV[1],
	MaxVarMV := MaxVarMV[1],
	DeadBand := DeadBand[1],
	MaxPV := MaxPV[1],
	MinPV := MinPV[1],
	Restart := Restart[1],
	SampleTime := 0.25,
	EnableP := TRUE,
	EnableI := TRUE,
	EnableD := TRUE,
	DerivPV := TRUE,
	Manual := Manual[1],
	Direct := FALSE,
	MeasureST := MeasureST,
	MV => PIDs.rPID_MV,
	EffST => EffST,
	Eff3ST => Eff3ST,
	MaxEffST => MaxEffST,
	MinEffST => MinEffST,
	ErrorCode => ErrorCodePID,	
	IntegralAction := IntegralAction
);

MV := PIDs.rPID_MV;

Restart[1] := false;

END_PROGRAM

// Device/Application/UserPOUs/Redundant/Recursividade
PROGRAM Recursividade
VAR
	Chamada1 : Delay;
	Chamada2 : Delay;
	Chamada3 : Delay;
	Chamada4 : Delay;
	Chamada5 : Delay;
	

END_VAR

// Esta POU existe para testar recursividade de TON,
// fato que apresentou problemas na alteração do compilador no passado
// FAÇA 2602


Chamada1();
Chamada2();
Chamada3();
Chamada4();
Chamada5();

Chamada1.tPT := T#1S;
Chamada2.tPT := T#1S;
Chamada3.tPT := T#1S;
Chamada4.tPT := T#1S;
Chamada5.tPT := T#1S;

Chamada1.bIN := NOT Chamada5.bQ;
Chamada2.bIN := Chamada1.bQ;
Chamada3.bIN := Chamada2.bQ;
Chamada4.bIN := Chamada3.bQ;
Chamada5.bIN := Chamada4.bQ;

END_PROGRAM

// Device/Application/UserFunctionsBlocks/Delay
FUNCTION_BLOCK Delay
VAR_INPUT
	bIN : BOOL;
	tPT : TIME;
END_VAR
VAR_OUTPUT
	tET : TIME;
	bQ : BOOL;
	
END_VAR
VAR
	t1: TON;	
	t2: Delay1;	
END_VAR

// Function Block que chama o TON para testar recursividade de TON que já apresentou problemas.
t1.IN:= bIN;
t1.PT:= tPT;
t1();
tET:= t1.ET;
bQ:= t1.Q;

// Function Block que chama outro Function Block
t2();

END_FUNCTION_BLOCK

// Device/Application/UserFunctionsBlocks/Delay1
FUNCTION_BLOCK Delay1
VAR_INPUT
	bInput : BOOL;
END_VAR
VAR_OUTPUT
	bOutput : BOOL;
END_VAR
VAR

END_VAR

// Apenas chamada de um outro Function Block

bOutput:= NOT bInput;

END_FUNCTION_BLOCK

// Device/Application/UserPOUs/Non-Redundant/CheckRedData
PROGRAM CheckRedData
VAR
	// Os limites dos laços, definidos a seguir, foram criados em função do bug 15023
	dwSizeS : DWORD;
	dwSizeQ : DWORD;
	dwSizeM : DWORD;
	dwSizeI : DWORD;
	iCheckValue : INT := 0;
	bStartup : BOOL := FALSE;
	dwIndexS : DWORD := 1;
	dwIndexQ : DWORD := 1;
	dwIndexM : DWORD := 1;
	dwIndexI : DWORD := 1;
	adwFailIndexSymb : ARRAY [0..100] OF DWORD;
	iReadValueSymb : ARRAY [0..100] OF INT;
	iExpectedValueSymb : ARRAY [0..100] OF INT;
	adwFailIndexSymb1 : ARRAY [0..100] OF DWORD;
	iReadValueSymb1 : ARRAY [0..100] OF INT;
	iExpectedValueSymb1 : ARRAY [0..100] OF INT;
	adwFailIndexSymb2 : ARRAY [0..100] OF DWORD;
	iReadValueSymb2 : ARRAY [0..100] OF INT;
	iExpectedValueSymb2 : ARRAY [0..100] OF INT;
	adwFailIndexSymb3 : ARRAY [0..100] OF DWORD;
	iReadValueSymb3 : ARRAY [0..100] OF INT;
	iExpectedValueSymb3 : ARRAY [0..100] OF INT;
	adwFailIndexSymb4 : ARRAY [0..100] OF DWORD;
	iReadValueSymb4 : ARRAY [0..100] OF INT;
	iExpectedValueSymb4 : ARRAY [0..100] OF INT;
	adwFailIndexQ : ARRAY [0..100] OF DWORD;
	iReadValueQ : ARRAY [0..100] OF INT;
	iExpectedValueQ : ARRAY [0..100] OF INT;
	adwFailIndexQ1 : ARRAY [0..100] OF DWORD;
	iReadValueQ1 : ARRAY [0..100] OF INT;
	iExpectedValueQ1 : ARRAY [0..100] OF INT;
	adwFailIndexM : ARRAY [0..100] OF DWORD;
	iReadValueM : ARRAY [0..100] OF INT;
	iExpectedValueM : ARRAY [0..100] OF INT;
	adwFailIndexM1 : ARRAY [0..100] OF DWORD;
	iReadValueM1 : ARRAY [0..100] OF INT;
	iExpectedValueM1 : ARRAY [0..100] OF INT;
	adwFailIndexI : ARRAY [0..100] OF DWORD;
	iReadValueI : ARRAY [0..100] OF INT;
	iExpectedValueI : ARRAY [0..100] OF INT;
	adwFailIndexI1 : ARRAY [0..100] OF DWORD;
	iReadValueI1 : ARRAY [0..100] OF INT;
	iExpectedValueI1 : ARRAY [0..100] OF INT;
	uliPouIniTime : ULINT;
	uliPouEndTime : ULINT;
END_VAR
VAR RETAIN
	iSyncFailCntS : INT := 0;
	iSyncFailCntS1 : INT := 0;
	iSyncFailCntS2: INT := 0;
	iSyncFailCntS3 : INT := 0;
	iSyncFailCntS4 : INT := 0;
	iSyncFailCntQ : INT := 0;
	iSyncFailCntQ1 : INT := 0;
	iSyncFailCntM : INT := 0;
	iSyncFailCntM1 : INT := 0;
	iSyncFailCntI : INT := 0;
	iSyncFailCntI1 : INT := 0;
END_VAR

// Registra o tempo do sistema
SysTimeGetUs(uliPouIniTime);

// Restaura variáveis na partida do sistema
IF bStartup = FALSE THEN
		NonRedPointer.piSSyncFailLoc^:= PersistentVars.iSyncFailCntSymb;
		NonRedPointer.piQSyncFailLoc^:= PersistentVars.iSyncFailCntQ;
		NonRedPointer.piMSyncFailLoc^:= PersistentVars.iSyncFailCntM;
		NonRedPointer.piISyncFailLoc^:= PersistentVars.iSyncFailCntI;
		
	// Inicializa os limites dos laços de verificação das variáveis redundantes
	dwSizeS:= (SIZEOF(Symbolics.aiRedundantArrayS)/SIZEOF(Symbolics.aiRedundantArrayS[1])) / ProjectConstants.dwCheckRedDataDivisor; 
	dwSizeQ:= (SIZEOF(ATs.aiRedundantArrayQ)/SIZEOF(ATs.aiRedundantArrayQ[1])) / ProjectConstants.dwCheckRedDataDivisor;
	dwSizeM:= (SIZEOF(ATs.aiRedundantArrayM)/SIZEOF(ATs.aiRedundantArrayM[1])) / ProjectConstants.dwCheckRedDataDivisor;
	dwSizeI:= (SIZEOF(ATs.aiRedundantArrayI)/SIZEOF(ATs.aiRedundantArrayI[1])) / ProjectConstants.dwCheckRedDataDivisor;
	// Indica que já inicializou as variáveis
	bStartup:= TRUE;
END_IF

// Reinicializa os contadores de falha, caso solicitado
IF SymbolicsNonRedundant.bEnableCleanStats_CheckRedData = TRUE THEN
	iSyncFailCntS:= 0;
	iSyncFailCntS1:= 0;
	iSyncFailCntS2:= 0;
	iSyncFailCntS3:= 0;
	iSyncFailCntS4:= 0;
	iSyncFailCntQ:= 0;
	iSyncFailCntQ1:= 0;
	iSyncFailCntM:= 0;
	iSyncFailCntM1:= 0;
	iSyncFailCntI:= 0;
	iSyncFailCntI1:= 0;
	SymbolicsNonRedundant.bEnableCleanStats_CheckRedData:= FALSE;
END_IF

// Se este PLC está no estado não-ativo e o outro no estado ativo, consiste os dados redundantes
IF DG_NX4010.tRedundancy.RedDgnLoc.sGeneral_Diag.eRedState <> REDUNDANCY_STATE.ACTIVE AND 
   DG_NX4010.tRedundancy.RedDgnRem.sGeneral_Diag.eRedState =  REDUNDANCY_STATE.ACTIVE THEN
	// Detecta necessidade de inicialização do valor dos dados redundantes
	IF iCheckValue = 0 THEN
		IF Symbolics.iValueRed >= ProjectConstants.iValueRedLimit THEN
			iCheckValue:= 1;
		ELSE
			iCheckValue:= Symbolics.iValueRed + 1;
		END_IF
	ELSE
		// Consistência do array simbólico
		WHILE dwIndexS <= dwSizeS DO
			IF iCheckValue <> Symbolics.aiRedundantArrayS[dwIndexS] OR iCheckValue <> Symbolics.aiRedundantArrayS1[dwIndexS] OR iCheckValue <> Symbolics.aiRedundantArrayS2[dwIndexS] OR iCheckValue <> Symbolics.aiRedundantArrayS3[dwIndexS] OR iCheckValue <> Symbolics.aiRedundantArrayS4[dwIndexS] THEN
				// Salva informações extras da falha: índice, valor lido e valor esperado
				IF iSyncFailCntS < 100 THEN
					adwFailIndexSymb[iSyncFailCntS]:= dwIndexS;
					iReadValueSymb[iSyncFailCntS]:= Symbolics.aiRedundantArrayS[dwIndexS];
					iExpectedValueSymb[iSyncFailCntS]:= iCheckValue;
				END_IF	
				IF iSyncFailCntS1 < 100 THEN
					adwFailIndexSymb1[iSyncFailCntS1]:= dwIndexS;
					iReadValueSymb1[iSyncFailCntS1]:= Symbolics.aiRedundantArrayS1[dwIndexS];
					iExpectedValueSymb1[iSyncFailCntS1]:= iCheckValue;
				END_IF	
				IF iSyncFailCntS2 < 100 THEN
					adwFailIndexSymb2[iSyncFailCntS2]:= dwIndexS;
					iReadValueSymb2[iSyncFailCntS2]:= Symbolics.aiRedundantArrayS2[dwIndexS];
					iExpectedValueSymb2[iSyncFailCntS2]:= iCheckValue;
				END_IF	
				IF iSyncFailCntS3 < 100 THEN
					adwFailIndexSymb3[iSyncFailCntS3]:= dwIndexS;
					iReadValueSymb3[iSyncFailCntS3]:= Symbolics.aiRedundantArrayS3[dwIndexS];
					iExpectedValueSymb3[iSyncFailCntS3]:= iCheckValue;
				END_IF	
				IF iSyncFailCntS4 < 100 THEN
					adwFailIndexSymb4[iSyncFailCntS4]:= dwIndexS;
					iReadValueSymb4[iSyncFailCntS4]:= Symbolics.aiRedundantArrayS4[dwIndexS];
					iExpectedValueSymb4[iSyncFailCntS4]:= iCheckValue;
				END_IF	
				// Incrementa o contador de falhas
				IF NonRedPointer.piSSyncFailLoc^ < ProjectConstants.iFailCounterLimit THEN							
				iSyncFailCntS:= iSyncFailCntS + 1;
				iSyncFailCntS1:= iSyncFailCntS1 + 1;
				iSyncFailCntS2:= iSyncFailCntS2 + 1;
				iSyncFailCntS3:= iSyncFailCntS3 + 1;
				iSyncFailCntS4:= iSyncFailCntS4 + 1;
				NonRedPointer.piSSyncFailLoc^:= iSyncFailCntS;
				END_IF
				EXIT;
			END_IF
			dwIndexS:= dwIndexS + 1;
		END_WHILE
		// Calcula próximo índice a ser consistido
		IF dwSizeS >= (SIZEOF(Symbolics.aiRedundantArrayS)/SIZEOF(Symbolics.aiRedundantArrayS[1])) THEN
			dwIndexS:= 1;
			dwSizeS:= (SIZEOF(Symbolics.aiRedundantArrayS)/SIZEOF(Symbolics.aiRedundantArrayS[1])) / ProjectConstants.dwCheckRedDataDivisor;
		ELSE
			dwIndexS:= dwSizeS;
			dwSizeS:= dwSizeS + (SIZEOF(Symbolics.aiRedundantArrayS)/SIZEOF(Symbolics.aiRedundantArrayS[1])) / ProjectConstants.dwCheckRedDataDivisor;
		END_IF
		
		// Consistência do array %Q
		WHILE dwIndexQ <= dwSizeQ DO
			IF iCheckValue <> ATs.aiRedundantArrayQ[dwIndexQ] OR iCheckValue <> ATs.aiRedundantArrayQ1[dwIndexQ] THEN
				// Salva informações extras da falha: índice, valor lido e valor esperado
				IF iSyncFailCntQ < 100 THEN
					adwFailIndexQ[iSyncFailCntQ]:= dwIndexQ;
					iReadValueQ[iSyncFailCntQ]:= ATs.aiRedundantArrayQ[dwIndexQ];
					iExpectedValueQ[iSyncFailCntQ]:= iCheckValue;		
				END_IF	
				IF iSyncFailCntQ1 < 100 THEN
					adwFailIndexQ1[iSyncFailCntQ1]:= dwIndexQ;
					iReadValueQ1[iSyncFailCntQ1]:= ATs.aiRedundantArrayQ1[dwIndexQ];
					iExpectedValueQ1[iSyncFailCntQ1]:= iCheckValue;		
				END_IF	
				// Incrementa o contador de falhas
				IF NonRedPointer.piQSyncFailLoc^ < ProjectConstants.iFailCounterLimit THEN		
				iSyncFailCntQ:= iSyncFailCntQ + 1;
				iSyncFailCntQ1:= iSyncFailCntQ1 + 1;
				NonRedPointer.piQSyncFailLoc^:= iSyncFailCntQ;
				END_IF
				EXIT;
			END_IF
			dwIndexQ:= dwIndexQ + 1;
		END_WHILE
		// Calcula próximo índice a ser consistido
		IF dwSizeQ >= (SIZEOF(ATs.aiRedundantArrayQ)/SIZEOF(ATs.aiRedundantArrayQ[1])) THEN
			dwIndexQ:= 1;
			dwSizeQ:= (SIZEOF(ATs.aiRedundantArrayQ)/SIZEOF(ATs.aiRedundantArrayQ[1])) / ProjectConstants.dwCheckRedDataDivisor;
		ELSE
			dwIndexQ:= dwSizeQ;
			dwSizeQ:= dwSizeQ + (SIZEOF(ATs.aiRedundantArrayQ)/SIZEOF(ATs.aiRedundantArrayQ[1])) / ProjectConstants.dwCheckRedDataDivisor;
		END_IF
		
		// Consistência do array %M
		WHILE dwIndexM <= dwSizeM DO
			IF iCheckValue <> ATs.aiRedundantArrayM[dwIndexM] OR iCheckValue <> ATs.aiRedundantArrayM1[dwIndexM]THEN
				// Salva informações extras da falha: índice, valor lido e valor esperado
				IF iSyncFailCntM < 100 THEN
					adwFailIndexM[iSyncFailCntM]:= dwIndexM;
					iReadValueM[iSyncFailCntM]:= ATs.aiRedundantArrayM[dwIndexM];
					iExpectedValueM[iSyncFailCntM]:=iCheckValue;
				END_IF
				IF iSyncFailCntM1 < 100 THEN
					adwFailIndexM1[iSyncFailCntM1]:= dwIndexM;
					iReadValueM1[iSyncFailCntM1]:= ATs.aiRedundantArrayM1[dwIndexM];
					iExpectedValueM1[iSyncFailCntM1]:=iCheckValue;
				END_IF
				// Incrementa o contador de falhas
				IF NonRedPointer.piMSyncFailLoc^ < ProjectConstants.iFailCounterLimit THEN									
				iSyncFailCntM:= iSyncFailCntM + 1;
				iSyncFailCntM1:= iSyncFailCntM1 + 1;
				NonRedPointer.piMSyncFailLoc^:= iSyncFailCntM;
				END_IF
				EXIT;
			END_IF
			dwIndexM:= dwIndexM + 1;
		END_WHILE
		// Calcula próximo índice a ser consistido
		IF dwSizeM >= (SIZEOF(ATs.aiRedundantArrayM)/SIZEOF(ATs.aiRedundantArrayM[1])) THEN
			dwIndexM:= 1;
			dwSizeM:= (SIZEOF(ATs.aiRedundantArrayM)/SIZEOF(ATs.aiRedundantArrayM[1])) / ProjectConstants.dwCheckRedDataDivisor;
		ELSE
			dwIndexM:= dwSizeM;
			dwSizeM:= dwSizeM + (SIZEOF(ATs.aiRedundantArrayM)/SIZEOF(ATs.aiRedundantArrayM[1])) / ProjectConstants.dwCheckRedDataDivisor;
		END_IF
		
		// Consistência do array %I
		WHILE dwIndexI <= dwSizeI DO
			IF iCheckValue <> ATs.aiRedundantArrayI[dwIndexI] OR iCheckValue <> ATs.aiRedundantArrayI1[dwIndexI] THEN
				// Salva informações extras da falha: índice, valor lido e valor esperado
				IF iSyncFailCntI < 100 THEN
					adwFailIndexI[iSyncFailCntI]:= dwIndexI;
					iReadValueI[iSyncFailCntI]:= ATs.aiRedundantArrayI[dwIndexI];
					iExpectedValueI[iSyncFailCntI]:= iCheckValue;
				END_IF	
				IF iSyncFailCntI1 < 100 THEN
					adwFailIndexI1[iSyncFailCntI1]:= dwIndexI;
					iReadValueI[iSyncFailCntI1]:= ATs.aiRedundantArrayI1[dwIndexI];
					iExpectedValueI1[iSyncFailCntI1]:= iCheckValue;
				END_IF	
				// Incrementa o contador de falhas
				IF NonRedPointer.piISyncFailLoc^ < ProjectConstants.iFailCounterLimit THEN				
				iSyncFailCntI:= iSyncFailCntI + 1;
				iSyncFailCntI1:= iSyncFailCntI1 + 1;
				NonRedPointer.piISyncFailLoc^:= iSyncFailCntI;
				END_IF
				EXIT;
			END_IF
			dwIndexI:= dwIndexI + 1;
		END_WHILE
		// Calcula próximo índice a ser consistido
		IF dwSizeI >= (SIZEOF(ATs.aiRedundantArrayI)/SIZEOF(ATs.aiRedundantArrayI[1])) THEN
			dwIndexI:= 1;
			dwSizeI:= (SIZEOF(ATs.aiRedundantArrayI)/SIZEOF(ATs.aiRedundantArrayI[1])) / ProjectConstants.dwCheckRedDataDivisor;
		ELSE
			dwIndexI:= dwSizeI;
			dwSizeI:= dwSizeI + (SIZEOF(ATs.aiRedundantArrayI)/SIZEOF(ATs.aiRedundantArrayI[1])) / ProjectConstants.dwCheckRedDataDivisor;
		END_IF
		
		// Incrementa o valor das variáveis redundantes
		IF Symbolics.iValueRed >= ProjectConstants.iValueRedLimit THEN
			iCheckValue:= 1;
		ELSE
			iCheckValue:= Symbolics.iValueRed + 1;
		END_IF
		
		// Registra o tempo do sistema
		SysTimeGetUs(uliPouEndTime);
		// Calcula duração mínima/máxima desta POU
		MinMaxTimes.uliPouMinTime_CheckRedData:= MIN(MinMaxTimes.uliPouMinTime_CheckRedData, uliPouEndTime - uliPouIniTime);
		MinMaxTimes.uliPouMaxTime_CheckRedData:= MAX(MinMaxTimes.uliPouMaxTime_CheckRedData, uliPouEndTime - uliPouIniTime);
	END_IF
ELSE
	// Incrementa o valor das variáveis redundantes
	IF Symbolics.iValueRed >= ProjectConstants.iValueRedLimit THEN
		iCheckValue:= 1;
	ELSE
		iCheckValue:= Symbolics.iValueRed + 1;
	END_IF
END_IF

END_PROGRAM

// Device/Application/UserPOUs/Non-Redundant/CycleTimes
PROGRAM CycleTimes
VAR
	sAppName : STRING;
	psAppName : POINTER TO STRING;
	bSetup : BOOL := TRUE;
	adwAvgMainTask : ARRAY [1..250] OF DWORD;
	adwAvgConfigTask : ARRAY [1..250] OF DWORD;
	dwMainTaskSum : DWORD := 0;
	dwConfigTaskSum : DWORD := 0;
	iMainIndex : INT := 1;
	iConfigIndex : INT := 1;
	uliPouIniTime : ULINT;
	uliPouEndTime : ULINT;
	// TRUE se algunm dos PLCs está ativo
	bPouActiveTime : BOOL;
END_VAR

// Registra os tempos de ciclo máximo, mínimo e médio das tarefas MainTask e Configuration do PLC no estado ATIVO

// Registra o tempo do sistema
SysTimeGetUs(uliPouIniTime);

// A principio nenhum PLC está ativo
bPouActiveTime:= FALSE;

IF bSetup = TRUE THEN
	sAppName:= 'Application';		// Variável recebe o nome da aplicação.
	psAppName:= ADR(sAppName);		// Ponteiro com o nome da aplicação.

	Task_Information.TI_MainTask.sTaskName := 'MainTask';
	Task_Information.TI_MainTask.psTaskName := ADR(Task_Information.TI_MainTask.sTaskName);
	Task_Information.TI_MainTask.pstTaskInfo := ADR (Task_Information.TI_MainTask.TaskInfo);
	
	Task_Information.TI_Configuration.sTaskName := 'Configuration';
	Task_Information.TI_Configuration.psTaskName := ADR(Task_Information.TI_Configuration.sTaskName);
	Task_Information.TI_Configuration.pstTaskInfo := ADR (Task_Information.TI_Configuration.TaskInfo);
	
	Task_Information.TI_MODBUS_Client_2.sTaskName := 'ATModbusMODBUS_Client_2';
	Task_Information.TI_MODBUS_Client_2.psTaskName := ADR(Task_Information.TI_MODBUS_Client_2.sTaskName);
	Task_Information.TI_MODBUS_Client_2.pstTaskInfo := ADR (Task_Information.TI_MODBUS_Client_2.TaskInfo);	
	
	Task_Information.TI_MODBUS_Client_3.sTaskName := 'ATModbusMODBUS_Client_3';
	Task_Information.TI_MODBUS_Client_3.psTaskName := ADR(Task_Information.TI_MODBUS_Client_3.sTaskName);
	Task_Information.TI_MODBUS_Client_3.pstTaskInfo := ADR (Task_Information.TI_MODBUS_Client_3.TaskInfo);
	
	Task_Information.TI_MODBUS_Master_1.sTaskName := 'ATModbusMODBUS_Master_1';
	Task_Information.TI_MODBUS_Master_1.psTaskName := ADR(Task_Information.TI_MODBUS_Master_1.sTaskName);
	Task_Information.TI_MODBUS_Master_1.pstTaskInfo := ADR (Task_Information.TI_MODBUS_Master_1.TaskInfo);
	
	Task_Information.TI_MODBUS_Server_2.sTaskName := 'ATModbusMODBUS_Server_2';
	Task_Information.TI_MODBUS_Server_2.psTaskName := ADR(Task_Information.TI_MODBUS_Server_2.sTaskName);
	Task_Information.TI_MODBUS_Server_2.pstTaskInfo := ADR (Task_Information.TI_MODBUS_Server_2.TaskInfo);
	
	Task_Information.TI_MODBUS_Server_3.sTaskName := 'ATModbusMODBUS_Server_3';
	Task_Information.TI_MODBUS_Server_3.psTaskName := ADR(Task_Information.TI_MODBUS_Server_3.sTaskName);
	Task_Information.TI_MODBUS_Server_3.pstTaskInfo := ADR (Task_Information.TI_MODBUS_Server_3.TaskInfo);
	
	Task_Information.TI_MODBUS_Slave_1.sTaskName := 'ATModbusMODBUS_Slave_1';
	Task_Information.TI_MODBUS_Slave_1.psTaskName := ADR(Task_Information.TI_MODBUS_Slave_1.sTaskName);
	Task_Information.TI_MODBUS_Slave_1.pstTaskInfo := ADR (Task_Information.TI_MODBUS_Slave_1.TaskInfo);

	bSetup:= FALSE;
END_IF

